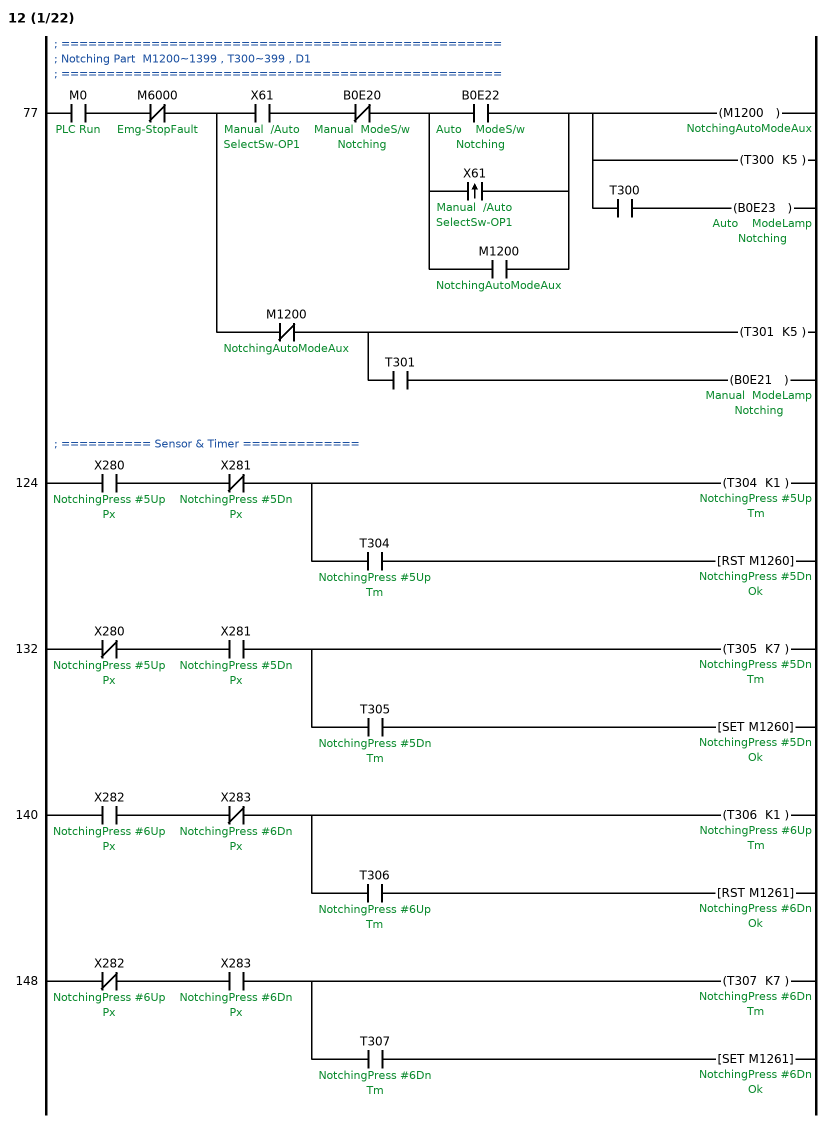
; =================================================
; Notching Part  M1200~1399 , T300~399 , D1
; =================================================
77    LD      M0  ; PLC Run
      ANI     M6000  ; Emg-StopFault
      MPS
      AND     X61  ; Manual  /Auto   SelectSw-OP1
      ANI     B0E20  ; Manual  ModeS/w Notching
      LD      B0E22  ; Auto    ModeS/w Notching
      ORP     X61  ; Manual  /Auto   SelectSw-OP1
      OR      M1200  ; NotchingAutoModeAux
      ANB
      OUT     M1200  ; NotchingAutoModeAux
      OUT     T300 K5
      AND     T300
      OUT     B0E23  ; Auto    ModeLampNotching
      MPP
      ANI     M1200  ; NotchingAutoModeAux
      OUT     T301 K5
      AND     T301
      OUT     B0E21  ; Manual  ModeLampNotching
; ========== Sensor & Timer =============
124   LD      X280  ; NotchingPress #5Up Px
      ANI     X281  ; NotchingPress #5Dn Px
      OUT     T304 K1  ; NotchingPress #5Up Tm
      AND     T304  ; NotchingPress #5Up Tm
      RST     M1260  ; NotchingPress #5Dn Ok
132   LDI     X280  ; NotchingPress #5Up Px
      AND     X281  ; NotchingPress #5Dn Px
      OUT     T305 K7  ; NotchingPress #5Dn Tm
      AND     T305  ; NotchingPress #5Dn Tm
      SET     M1260  ; NotchingPress #5Dn Ok
140   LD      X282  ; NotchingPress #6Up Px
      ANI     X283  ; NotchingPress #6Dn Px
      OUT     T306 K1  ; NotchingPress #6Up Tm
      AND     T306  ; NotchingPress #6Up Tm
      RST     M1261  ; NotchingPress #6Dn Ok
148   LDI     X282  ; NotchingPress #6Up Px
      AND     X283  ; NotchingPress #6Dn Px
      OUT     T307 K7  ; NotchingPress #6Dn Tm
      AND     T307  ; NotchingPress #6Dn Tm
      SET     M1261  ; NotchingPress #6Dn Ok
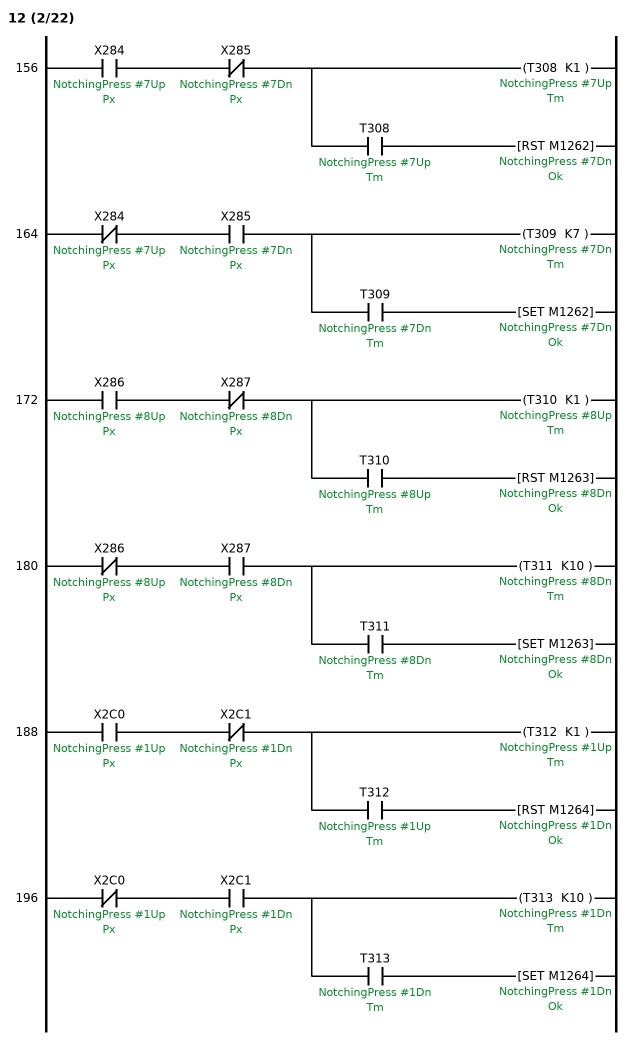
156   LD      X284  ; NotchingPress #7Up Px
      ANI     X285  ; NotchingPress #7Dn Px
      OUT     T308 K1  ; NotchingPress #7Up Tm
      AND     T308  ; NotchingPress #7Up Tm
      RST     M1262  ; NotchingPress #7Dn Ok
164   LDI     X284  ; NotchingPress #7Up Px
      AND     X285  ; NotchingPress #7Dn Px
      OUT     T309 K7  ; NotchingPress #7Dn Tm
      AND     T309  ; NotchingPress #7Dn Tm
      SET     M1262  ; NotchingPress #7Dn Ok
172   LD      X286  ; NotchingPress #8Up Px
      ANI     X287  ; NotchingPress #8Dn Px
      OUT     T310 K1  ; NotchingPress #8Up Tm
      AND     T310  ; NotchingPress #8Up Tm
      RST     M1263  ; NotchingPress #8Dn Ok
180   LDI     X286  ; NotchingPress #8Up Px
      AND     X287  ; NotchingPress #8Dn Px
      OUT     T311 K10  ; NotchingPress #8Dn Tm
      AND     T311  ; NotchingPress #8Dn Tm
      SET     M1263  ; NotchingPress #8Dn Ok
188   LD      X2C0  ; NotchingPress #1Up Px
      ANI     X2C1  ; NotchingPress #1Dn Px
      OUT     T312 K1  ; NotchingPress #1Up Tm
      AND     T312  ; NotchingPress #1Up Tm
      RST     M1264  ; NotchingPress #1Dn Ok
196   LDI     X2C0  ; NotchingPress #1Up Px
      AND     X2C1  ; NotchingPress #1Dn Px
      OUT     T313 K10  ; NotchingPress #1Dn Tm
      AND     T313  ; NotchingPress #1Dn Tm
      SET     M1264  ; NotchingPress #1Dn Ok
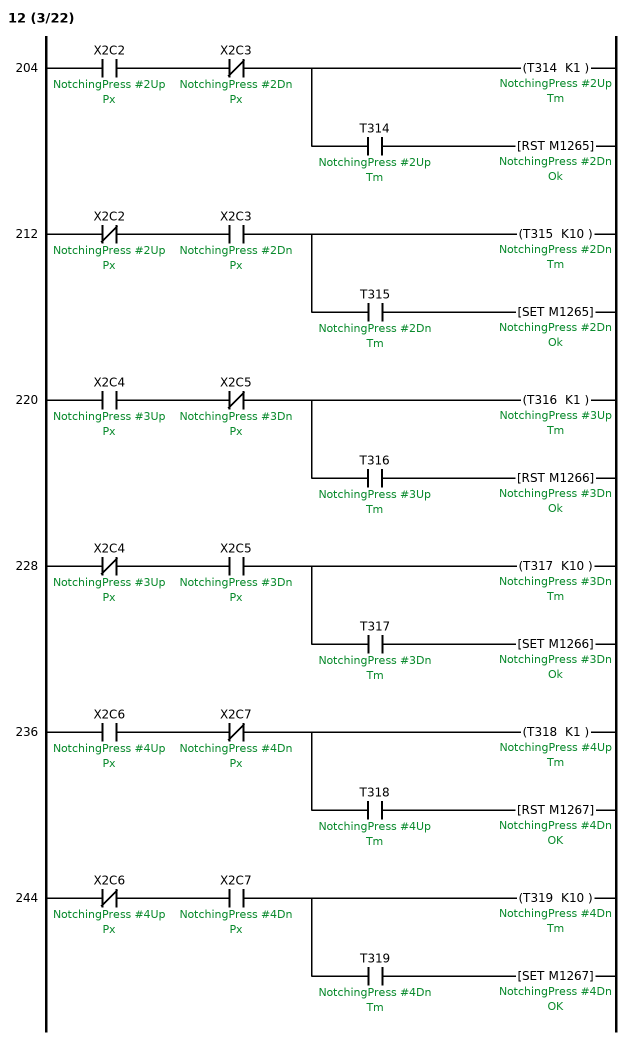
204   LD      X2C2  ; NotchingPress #2Up Px
      ANI     X2C3  ; NotchingPress #2Dn Px
      OUT     T314 K1  ; NotchingPress #2Up Tm
      AND     T314  ; NotchingPress #2Up Tm
      RST     M1265  ; NotchingPress #2Dn Ok
212   LDI     X2C2  ; NotchingPress #2Up Px
      AND     X2C3  ; NotchingPress #2Dn Px
      OUT     T315 K10  ; NotchingPress #2Dn Tm
      AND     T315  ; NotchingPress #2Dn Tm
      SET     M1265  ; NotchingPress #2Dn Ok
220   LD      X2C4  ; NotchingPress #3Up Px
      ANI     X2C5  ; NotchingPress #3Dn Px
      OUT     T316 K1  ; NotchingPress #3Up Tm
      AND     T316  ; NotchingPress #3Up Tm
      RST     M1266  ; NotchingPress #3Dn Ok
228   LDI     X2C4  ; NotchingPress #3Up Px
      AND     X2C5  ; NotchingPress #3Dn Px
      OUT     T317 K10  ; NotchingPress #3Dn Tm
      AND     T317  ; NotchingPress #3Dn Tm
      SET     M1266  ; NotchingPress #3Dn Ok
236   LD      X2C6  ; NotchingPress #4Up Px
      ANI     X2C7  ; NotchingPress #4Dn Px
      OUT     T318 K1  ; NotchingPress #4Up Tm
      AND     T318  ; NotchingPress #4Up Tm
      RST     M1267  ; NotchingPress #4Dn OK
244   LDI     X2C6  ; NotchingPress #4Up Px
      AND     X2C7  ; NotchingPress #4Dn Px
      OUT     T319 K10  ; NotchingPress #4Dn Tm
      AND     T319  ; NotchingPress #4Dn Tm
      SET     M1267  ; NotchingPress #4Dn OK
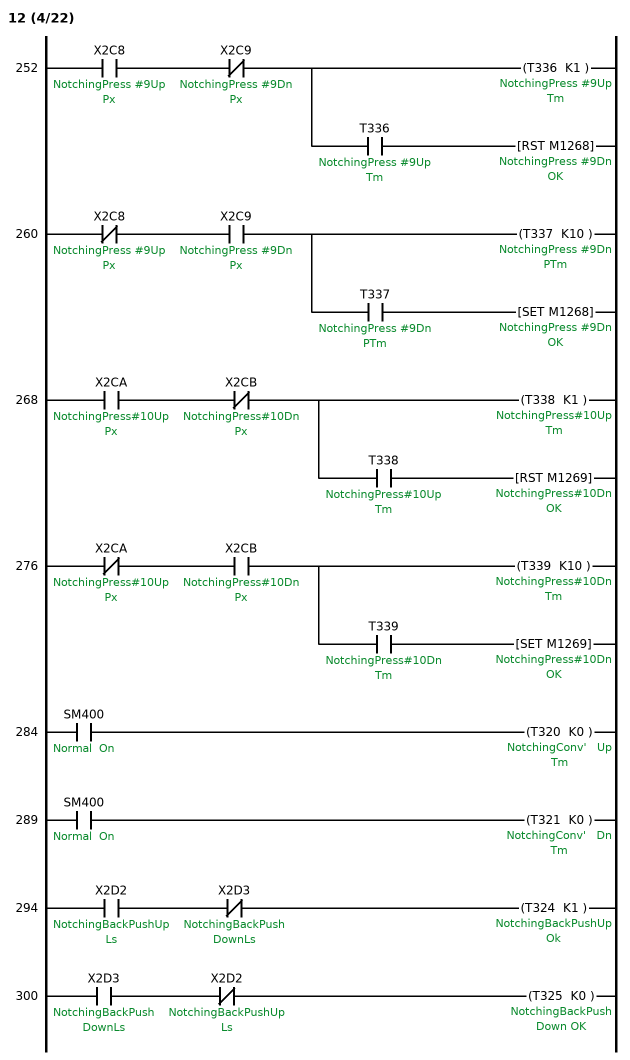
252   LD      X2C8  ; NotchingPress #9Up Px
      ANI     X2C9  ; NotchingPress #9Dn Px
      OUT     T336 K1  ; NotchingPress #9Up Tm
      AND     T336  ; NotchingPress #9Up Tm
      RST     M1268  ; NotchingPress #9Dn OK
260   LDI     X2C8  ; NotchingPress #9Up Px
      AND     X2C9  ; NotchingPress #9Dn Px
      OUT     T337 K10  ; NotchingPress #9Dn PTm
      AND     T337  ; NotchingPress #9Dn PTm
      SET     M1268  ; NotchingPress #9Dn OK
268   LD      X2CA  ; NotchingPress#10Up Px
      ANI     X2CB  ; NotchingPress#10Dn Px
      OUT     T338 K1  ; NotchingPress#10Up Tm
      AND     T338  ; NotchingPress#10Up Tm
      RST     M1269  ; NotchingPress#10Dn OK
276   LDI     X2CA  ; NotchingPress#10Up Px
      AND     X2CB  ; NotchingPress#10Dn Px
      OUT     T339 K10  ; NotchingPress#10Dn Tm
      AND     T339  ; NotchingPress#10Dn Tm
      SET     M1269  ; NotchingPress#10Dn OK
284   LD      SM400  ; Normal  On
      OUT     T320 K0  ; NotchingConv'   Up Tm
289   LD      SM400  ; Normal  On
      OUT     T321 K0  ; NotchingConv'   Dn Tm
294   LD      X2D2  ; NotchingBackPushUpLs
      ANI     X2D3  ; NotchingBackPushDownLs
      OUT     T324 K1  ; NotchingBackPushUp Ok
300   LD      X2D3  ; NotchingBackPushDownLs
      ANI     X2D2  ; NotchingBackPushUpLs
      OUT     T325 K0  ; NotchingBackPushDown OK
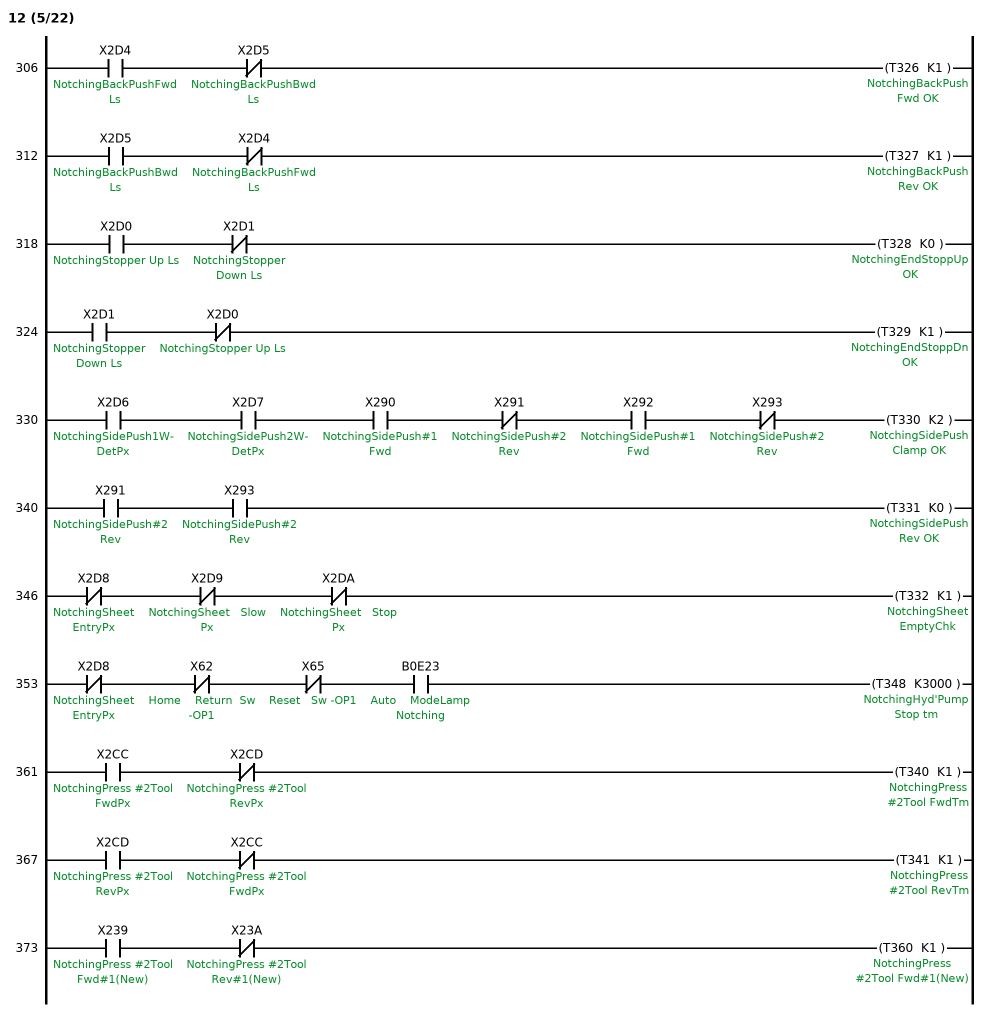
306   LD      X2D4  ; NotchingBackPushFwdLs
      ANI     X2D5  ; NotchingBackPushBwdLs
      OUT     T326 K1  ; NotchingBackPushFwd OK
312   LD      X2D5  ; NotchingBackPushBwdLs
      ANI     X2D4  ; NotchingBackPushFwdLs
      OUT     T327 K1  ; NotchingBackPushRev OK
318   LD      X2D0  ; NotchingStopper Up Ls
      ANI     X2D1  ; NotchingStopper Down Ls
      OUT     T328 K0  ; NotchingEndStoppUp OK
324   LD      X2D1  ; NotchingStopper Down Ls
      ANI     X2D0  ; NotchingStopper Up Ls
      OUT     T329 K1  ; NotchingEndStoppDn OK
330   LD      X2D6  ; NotchingSidePush1W-DetPx
      AND     X2D7  ; NotchingSidePush2W-DetPx
      AND     X290  ; NotchingSidePush#1 Fwd
      ANI     X291  ; NotchingSidePush#2 Rev
      AND     X292  ; NotchingSidePush#1 Fwd
      ANI     X293  ; NotchingSidePush#2 Rev
      OUT     T330 K2  ; NotchingSidePushClamp OK
340   LD      X291  ; NotchingSidePush#2 Rev
      AND     X293  ; NotchingSidePush#2 Rev
      OUT     T331 K0  ; NotchingSidePushRev OK
346   LDI     X2D8  ; NotchingSheet   EntryPx
      ANI     X2D9  ; NotchingSheet   Slow Px
      ANI     X2DA  ; NotchingSheet   Stop Px
      OUT     T332 K1  ; NotchingSheet   EmptyChk
353   LDI     X2D8  ; NotchingSheet   EntryPx
      ANI     X62  ; Home    Return  Sw -OP1
      ANI     X65  ; Reset   Sw -OP1
      AND     B0E23  ; Auto    ModeLampNotching
      OUT     T348 K3000  ; NotchingHyd'PumpStop tm
361   LD      X2CC  ; NotchingPress #2Tool FwdPx
      ANI     X2CD  ; NotchingPress #2Tool RevPx
      OUT     T340 K1  ; NotchingPress #2Tool FwdTm
367   LD      X2CD  ; NotchingPress #2Tool RevPx
      ANI     X2CC  ; NotchingPress #2Tool FwdPx
      OUT     T341 K1  ; NotchingPress #2Tool RevTm
373   LD      X239  ; NotchingPress #2Tool Fwd#1(New)
      ANI     X23A  ; NotchingPress #2Tool Rev#1(New)
      OUT     T360 K1  ; NotchingPress #2Tool Fwd#1(New)
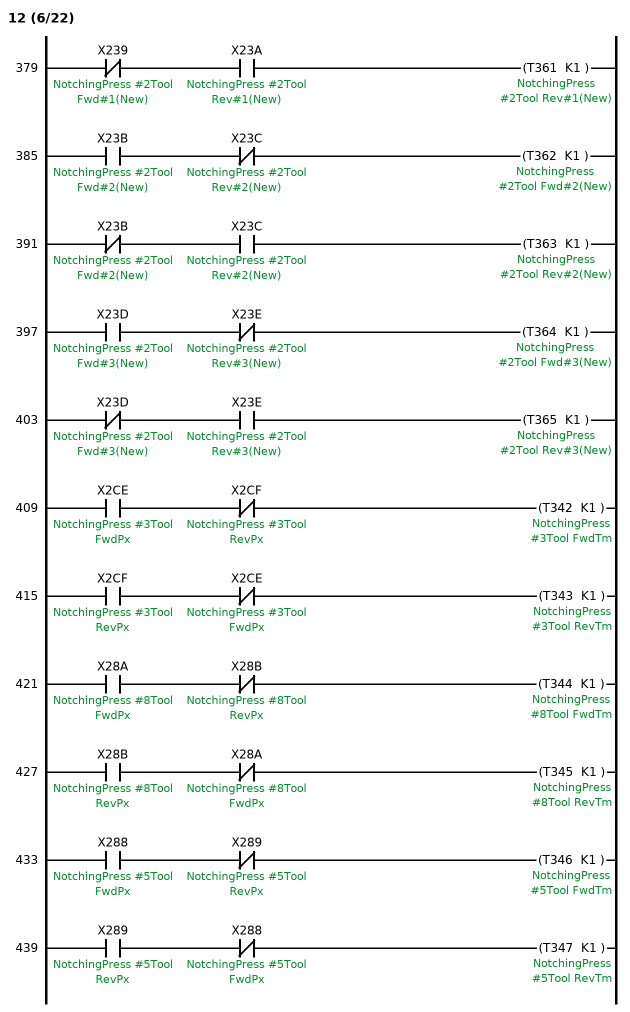
379   LDI     X239  ; NotchingPress #2Tool Fwd#1(New)
      AND     X23A  ; NotchingPress #2Tool Rev#1(New)
      OUT     T361 K1  ; NotchingPress #2Tool Rev#1(New)
385   LD      X23B  ; NotchingPress #2Tool Fwd#2(New)
      ANI     X23C  ; NotchingPress #2Tool Rev#2(New)
      OUT     T362 K1  ; NotchingPress #2Tool Fwd#2(New)
391   LDI     X23B  ; NotchingPress #2Tool Fwd#2(New)
      AND     X23C  ; NotchingPress #2Tool Rev#2(New)
      OUT     T363 K1  ; NotchingPress #2Tool Rev#2(New)
397   LD      X23D  ; NotchingPress #2Tool Fwd#3(New)
      ANI     X23E  ; NotchingPress #2Tool Rev#3(New)
      OUT     T364 K1  ; NotchingPress #2Tool Fwd#3(New)
403   LDI     X23D  ; NotchingPress #2Tool Fwd#3(New)
      AND     X23E  ; NotchingPress #2Tool Rev#3(New)
      OUT     T365 K1  ; NotchingPress #2Tool Rev#3(New)
409   LD      X2CE  ; NotchingPress #3Tool FwdPx
      ANI     X2CF  ; NotchingPress #3Tool RevPx
      OUT     T342 K1  ; NotchingPress #3Tool FwdTm
415   LD      X2CF  ; NotchingPress #3Tool RevPx
      ANI     X2CE  ; NotchingPress #3Tool FwdPx
      OUT     T343 K1  ; NotchingPress #3Tool RevTm
421   LD      X28A  ; NotchingPress #8Tool FwdPx
      ANI     X28B  ; NotchingPress #8Tool RevPx
      OUT     T344 K1  ; NotchingPress #8Tool FwdTm
427   LD      X28B  ; NotchingPress #8Tool RevPx
      ANI     X28A  ; NotchingPress #8Tool FwdPx
      OUT     T345 K1  ; NotchingPress #8Tool RevTm
433   LD      X288  ; NotchingPress #5Tool FwdPx
      ANI     X289  ; NotchingPress #5Tool RevPx
      OUT     T346 K1  ; NotchingPress #5Tool FwdTm
439   LD      X289  ; NotchingPress #5Tool RevPx
      ANI     X288  ; NotchingPress #5Tool FwdPx
      OUT     T347 K1  ; NotchingPress #5Tool RevTm
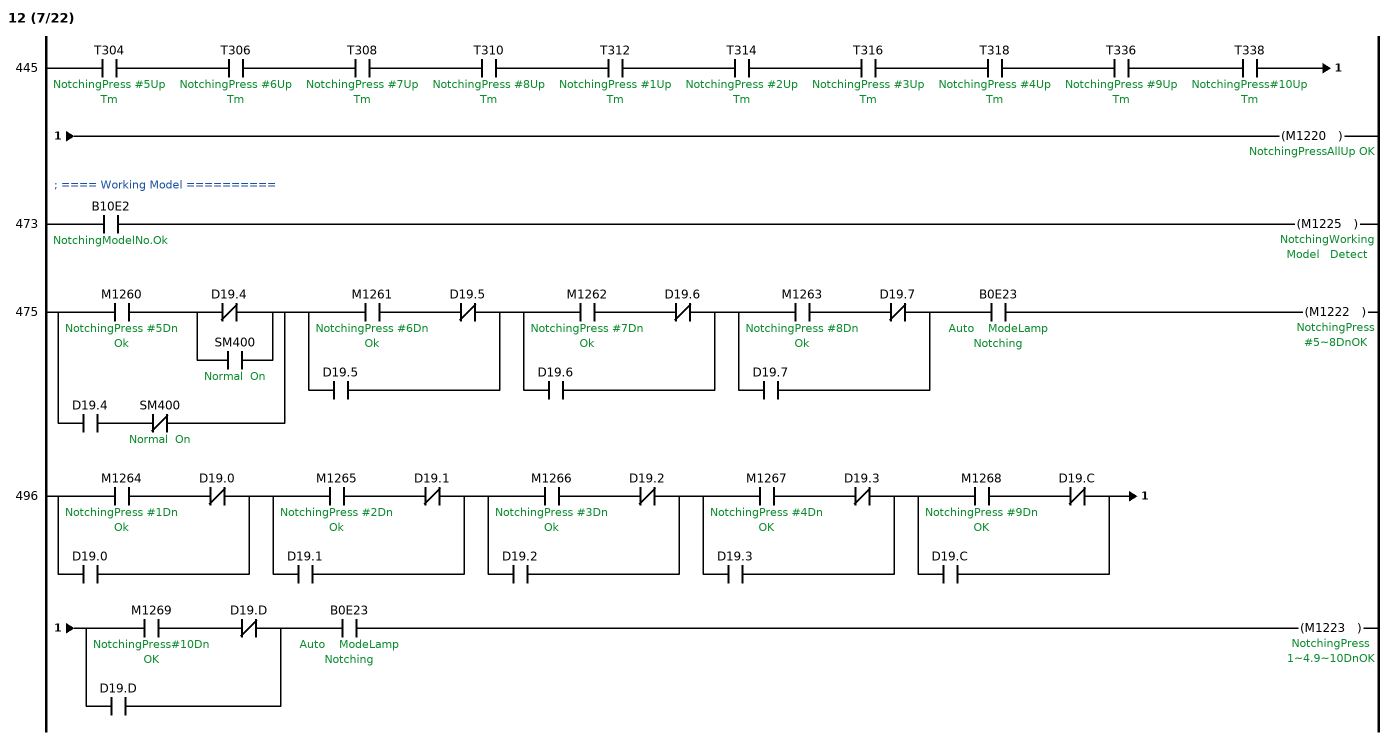
445   LD      T304  ; NotchingPress #5Up Tm
      AND     T306  ; NotchingPress #6Up Tm
      AND     T308  ; NotchingPress #7Up Tm
      AND     T310  ; NotchingPress #8Up Tm
      AND     T312  ; NotchingPress #1Up Tm
      AND     T314  ; NotchingPress #2Up Tm
      AND     T316  ; NotchingPress #3Up Tm
      AND     T318  ; NotchingPress #4Up Tm
      AND     T336  ; NotchingPress #9Up Tm
      AND     T338  ; NotchingPress#10Up Tm
      OUT     M1220  ; NotchingPressAllUp OK
; ==== Working Model ==========
473   LD      B10E2  ; NotchingModelNo.Ok
      OUT     M1225  ; NotchingWorking Model   Detect
475   LD      M1260  ; NotchingPress #5Dn Ok
      LDI     D19.4
      OR      SM400  ; Normal  On
      ANB
      LD      D19.4
      ANI     SM400  ; Normal  On
      ORB
      LD      M1261  ; NotchingPress #6Dn Ok
      ANI     D19.5
      OR      D19.5
      ANB
      LD      M1262  ; NotchingPress #7Dn Ok
      ANI     D19.6
      OR      D19.6
      ANB
      LD      M1263  ; NotchingPress #8Dn Ok
      ANI     D19.7
      OR      D19.7
      ANB
      AND     B0E23  ; Auto    ModeLampNotching
      OUT     M1222  ; NotchingPress   #5~8DnOK
496   LD      M1264  ; NotchingPress #1Dn Ok
      ANI     D19.0
      OR      D19.0
      LD      M1265  ; NotchingPress #2Dn Ok
      ANI     D19.1
      OR      D19.1
      ANB
      LD      M1266  ; NotchingPress #3Dn Ok
      ANI     D19.2
      OR      D19.2
      ANB
      LD      M1267  ; NotchingPress #4Dn OK
      ANI     D19.3
      OR      D19.3
      ANB
      LD      M1268  ; NotchingPress #9Dn OK
      ANI     D19.C
      OR      D19.C
      ANB
      LD      M1269  ; NotchingPress#10Dn OK
      ANI     D19.D
      OR      D19.D
      ANB
      AND     B0E23  ; Auto    ModeLampNotching
      OUT     M1223  ; NotchingPress   1~4.9~10DnOK
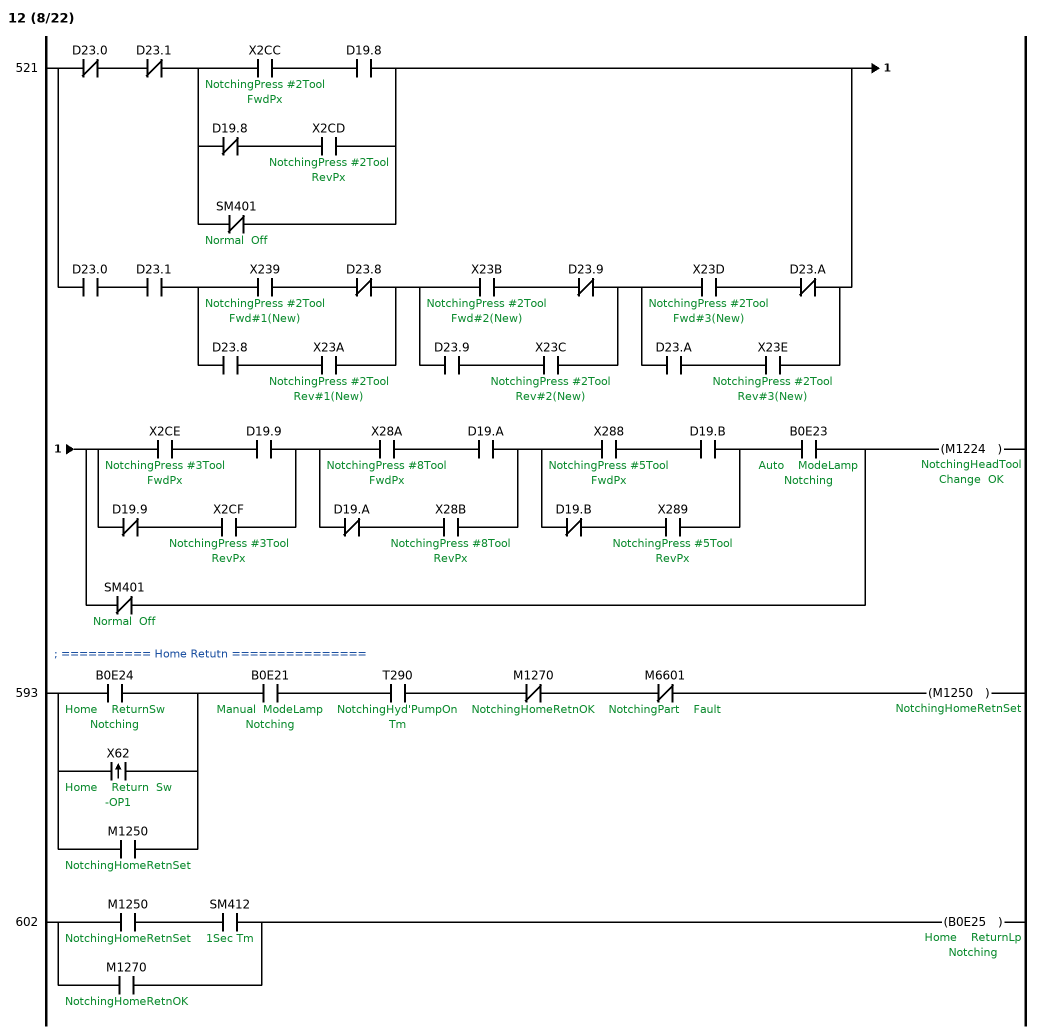
521   LDI     D23.0
      ANI     D23.1
      LD      X2CC  ; NotchingPress #2Tool FwdPx
      AND     D19.8
      LDI     D19.8
      AND     X2CD  ; NotchingPress #2Tool RevPx
      ORB
      ORI     SM401  ; Normal  Off
      ANB
      LD      D23.0
      AND     D23.1
      LD      X239  ; NotchingPress #2Tool Fwd#1(New)
      ANI     D23.8
      LD      D23.8
      AND     X23A  ; NotchingPress #2Tool Rev#1(New)
      ORB
      ANB
      LD      X23B  ; NotchingPress #2Tool Fwd#2(New)
      ANI     D23.9
      LD      D23.9
      AND     X23C  ; NotchingPress #2Tool Rev#2(New)
      ORB
      ANB
      LD      X23D  ; NotchingPress #2Tool Fwd#3(New)
      ANI     D23.A
      LD      D23.A
      AND     X23E  ; NotchingPress #2Tool Rev#3(New)
      ORB
      ANB
      ORB
      LD      X2CE  ; NotchingPress #3Tool FwdPx
      AND     D19.9
      LDI     D19.9
      AND     X2CF  ; NotchingPress #3Tool RevPx
      ORB
      LD      X28A  ; NotchingPress #8Tool FwdPx
      AND     D19.A
      LDI     D19.A
      AND     X28B  ; NotchingPress #8Tool RevPx
      ORB
      ANB
      LD      X288  ; NotchingPress #5Tool FwdPx
      AND     D19.B
      LDI     D19.B
      AND     X289  ; NotchingPress #5Tool RevPx
      ORB
      ANB
      AND     B0E23  ; Auto    ModeLampNotching
      ORI     SM401  ; Normal  Off
      ANB
      OUT     M1224  ; NotchingHeadToolChange  OK
; ========== Home Retutn ===============
593   LD      B0E24  ; Home    ReturnSwNotching
      ORP     X62  ; Home    Return  Sw -OP1
      OR      M1250  ; NotchingHomeRetnSet
      AND     B0E21  ; Manual  ModeLampNotching
      AND     T290  ; NotchingHyd'PumpOn Tm
      ANI     M1270  ; NotchingHomeRetnOK
      ANI     M6601  ; NotchingPart    Fault
      OUT     M1250  ; NotchingHomeRetnSet
602   LD      M1250  ; NotchingHomeRetnSet
      AND     SM412  ; 1Sec Tm
      OR      M1270  ; NotchingHomeRetnOK
      OUT     B0E25  ; Home    ReturnLpNotching
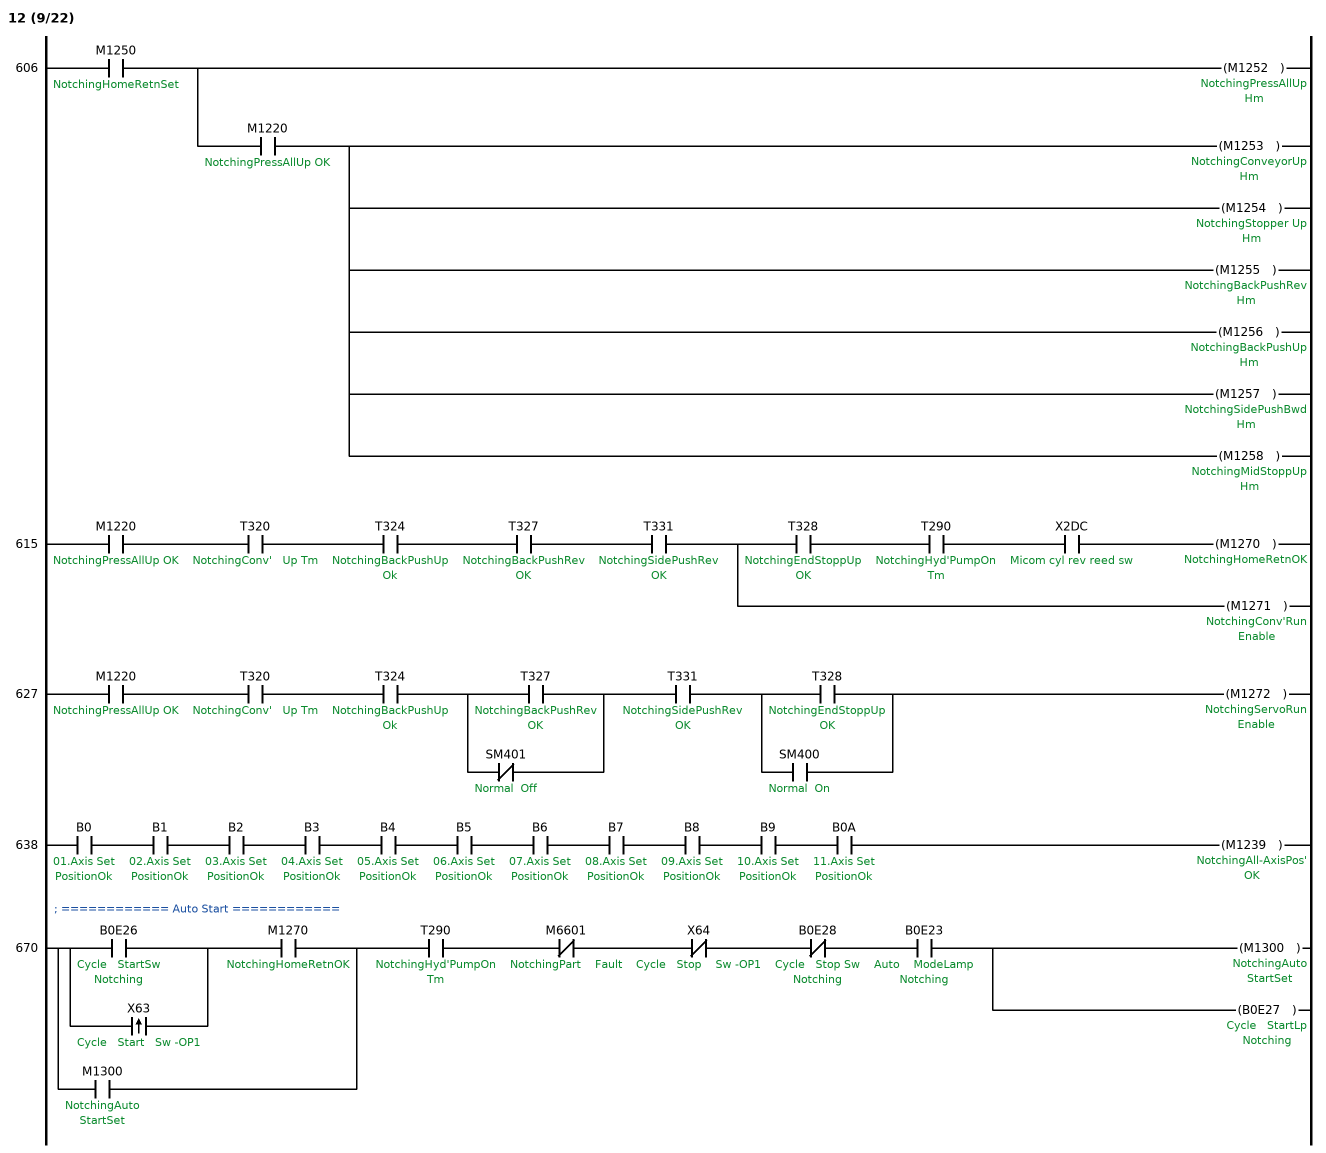
606   LD      M1250  ; NotchingHomeRetnSet
      OUT     M1252  ; NotchingPressAllUp Hm
      AND     M1220  ; NotchingPressAllUp OK
      OUT     M1253  ; NotchingConveyorUp Hm
      OUT     M1254  ; NotchingStopper Up Hm
      OUT     M1255  ; NotchingBackPushRev Hm
      OUT     M1256  ; NotchingBackPushUp Hm
      OUT     M1257  ; NotchingSidePushBwd Hm
      OUT     M1258  ; NotchingMidStoppUp Hm
615   LD      M1220  ; NotchingPressAllUp OK
      AND     T320  ; NotchingConv'   Up Tm
      AND     T324  ; NotchingBackPushUp Ok
      AND     T327  ; NotchingBackPushRev OK
      AND     T331  ; NotchingSidePushRev OK
      MPS
      AND     T328  ; NotchingEndStoppUp OK
      AND     T290  ; NotchingHyd'PumpOn Tm
      AND     X2DC  ; Micom cyl rev reed sw
      OUT     M1270  ; NotchingHomeRetnOK
      MPP
      OUT     M1271  ; NotchingConv'RunEnable
627   LD      M1220  ; NotchingPressAllUp OK
      AND     T320  ; NotchingConv'   Up Tm
      AND     T324  ; NotchingBackPushUp Ok
      LD      T327  ; NotchingBackPushRev OK
      ORI     SM401  ; Normal  Off
      ANB
      AND     T331  ; NotchingSidePushRev OK
      LD      T328  ; NotchingEndStoppUp OK
      OR      SM400  ; Normal  On
      ANB
      OUT     M1272  ; NotchingServoRunEnable
638   LD      B0  ; 01.Axis Set     PositionOk
      AND     B1  ; 02.Axis Set     PositionOk
      AND     B2  ; 03.Axis Set     PositionOk
      AND     B3  ; 04.Axis Set     PositionOk
      AND     B4  ; 05.Axis Set     PositionOk
      AND     B5  ; 06.Axis Set     PositionOk
      AND     B6  ; 07.Axis Set     PositionOk
      AND     B7  ; 08.Axis Set     PositionOk
      AND     B8  ; 09.Axis Set     PositionOk
      AND     B9  ; 10.Axis Set     PositionOk
      AND     B0A  ; 11.Axis Set     PositionOk
      OUT     M1239  ; NotchingAll-AxisPos' OK
; ============ Auto Start ============
670   LD      B0E26  ; Cycle   StartSw Notching
      ORP     X63  ; Cycle   Start   Sw -OP1
      AND     M1270  ; NotchingHomeRetnOK
      OR      M1300  ; NotchingAuto    StartSet
      AND     T290  ; NotchingHyd'PumpOn Tm
      ANI     M6601  ; NotchingPart    Fault
      ANI     X64  ; Cycle   Stop    Sw -OP1
      ANI     B0E28  ; Cycle   Stop Sw Notching
      AND     B0E23  ; Auto    ModeLampNotching
      OUT     M1300  ; NotchingAuto    StartSet
      OUT     B0E27  ; Cycle   StartLp Notching
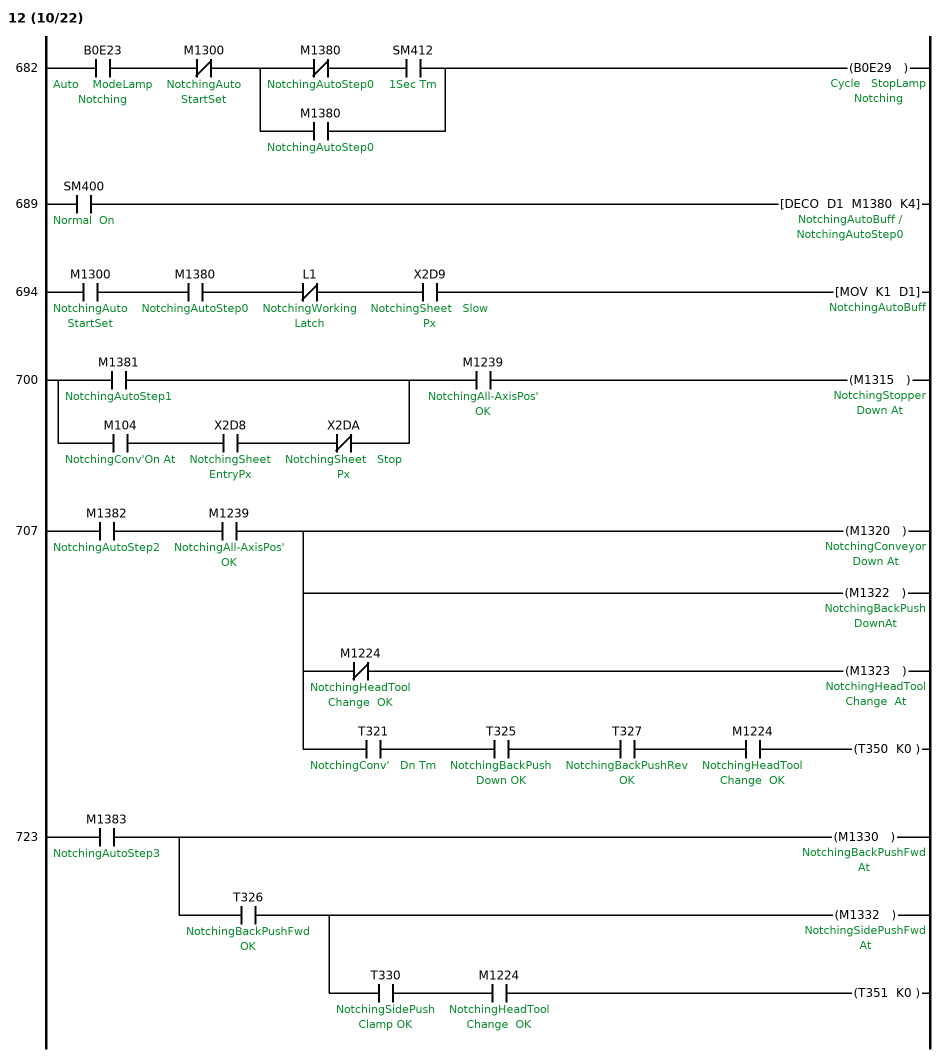
682   LD      B0E23  ; Auto    ModeLampNotching
      ANI     M1300  ; NotchingAuto    StartSet
      LDI     M1380  ; NotchingAutoStep0
      AND     SM412  ; 1Sec Tm
      OR      M1380  ; NotchingAutoStep0
      ANB
      OUT     B0E29  ; Cycle   StopLampNotching
689   LD      SM400  ; Normal  On
      DECO    D1 M1380 K4  ; NotchingAutoBuff
694   LD      M1300  ; NotchingAuto    StartSet
      AND     M1380  ; NotchingAutoStep0
      ANI     L1  ; NotchingWorking Latch
      AND     X2D9  ; NotchingSheet   Slow Px
      MOV     K1 D1
700   LD      M1381  ; NotchingAutoStep1
      LD      M104  ; NotchingConv'On At
      AND     X2D8  ; NotchingSheet   EntryPx
      ANI     X2DA  ; NotchingSheet   Stop Px
      ORB
      AND     M1239  ; NotchingAll-AxisPos' OK
      OUT     M1315  ; NotchingStopper Down At
707   LD      M1382  ; NotchingAutoStep2
      AND     M1239  ; NotchingAll-AxisPos' OK
      OUT     M1320  ; NotchingConveyorDown At
      OUT     M1322  ; NotchingBackPushDownAt
      MPS
      ANI     M1224  ; NotchingHeadToolChange  OK
      OUT     M1323  ; NotchingHeadToolChange  At
      MPP
      AND     T321  ; NotchingConv'   Dn Tm
      AND     T325  ; NotchingBackPushDown OK
      AND     T327  ; NotchingBackPushRev OK
      AND     M1224  ; NotchingHeadToolChange  OK
      OUT     T350 K0
723   LD      M1383  ; NotchingAutoStep3
      OUT     M1330  ; NotchingBackPushFwdAt
      AND     T326  ; NotchingBackPushFwd OK
      OUT     M1332  ; NotchingSidePushFwdAt
      AND     T330  ; NotchingSidePushClamp OK
      AND     M1224  ; NotchingHeadToolChange  OK
      OUT     T351 K0
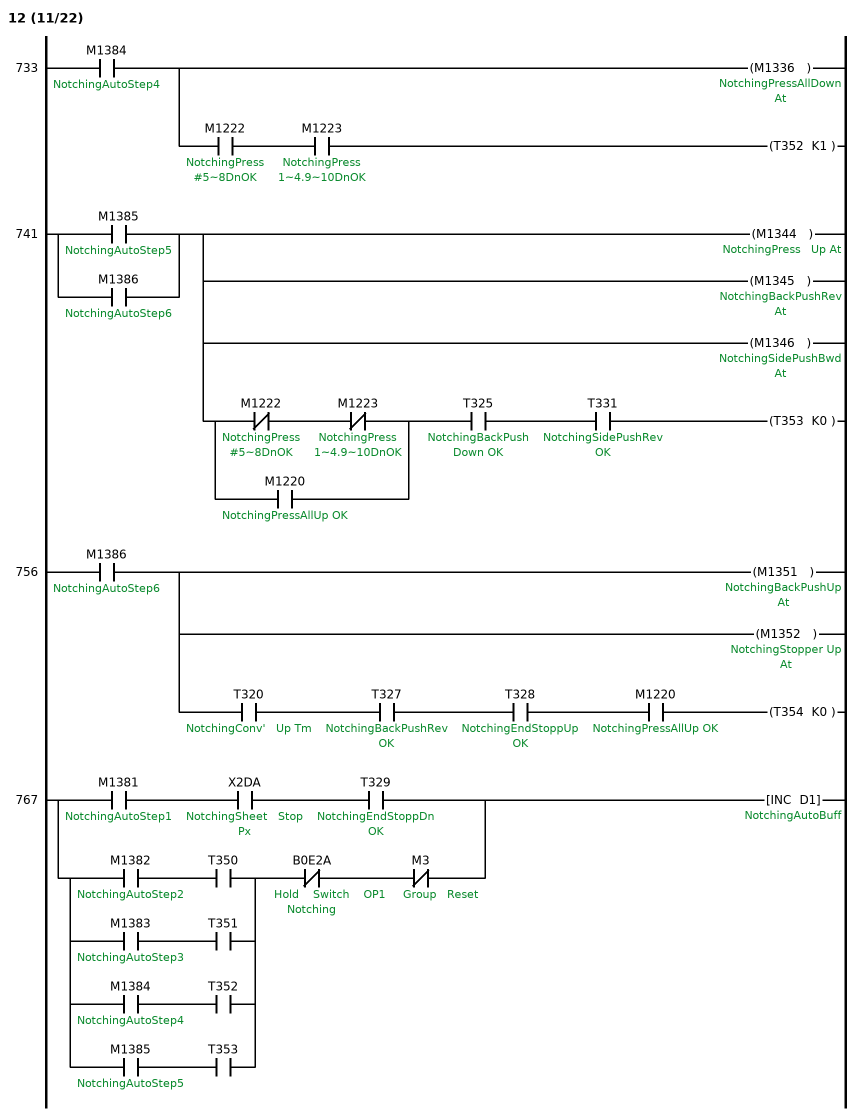
733   LD      M1384  ; NotchingAutoStep4
      OUT     M1336  ; NotchingPressAllDown At
      AND     M1222  ; NotchingPress   #5~8DnOK
      AND     M1223  ; NotchingPress   1~4.9~10DnOK
      OUT     T352 K1
741   LD      M1385  ; NotchingAutoStep5
      OR      M1386  ; NotchingAutoStep6
      OUT     M1344  ; NotchingPress   Up At
      OUT     M1345  ; NotchingBackPushRev At
      OUT     M1346  ; NotchingSidePushBwd At
      LDI     M1222  ; NotchingPress   #5~8DnOK
      ANI     M1223  ; NotchingPress   1~4.9~10DnOK
      OR      M1220  ; NotchingPressAllUp OK
      ANB
      AND     T325  ; NotchingBackPushDown OK
      AND     T331  ; NotchingSidePushRev OK
      OUT     T353 K0
756   LD      M1386  ; NotchingAutoStep6
      OUT     M1351  ; NotchingBackPushUp At
      OUT     M1352  ; NotchingStopper Up At
      AND     T320  ; NotchingConv'   Up Tm
      AND     T327  ; NotchingBackPushRev OK
      AND     T328  ; NotchingEndStoppUp OK
      AND     M1220  ; NotchingPressAllUp OK
      OUT     T354 K0
767   LD      M1381  ; NotchingAutoStep1
      AND     X2DA  ; NotchingSheet   Stop Px
      AND     T329  ; NotchingEndStoppDn OK
      LD      M1382  ; NotchingAutoStep2
      AND     T350
      LD      M1383  ; NotchingAutoStep3
      AND     T351
      ORB
      LD      M1384  ; NotchingAutoStep4
      AND     T352
      ORB
      LD      M1385  ; NotchingAutoStep5
      AND     T353
      ORB
      ANI     B0E2A  ; Hold    Switch  Notching
      ANI     M3  ; OP1     Group   Reset
      ORB
      INC     D1
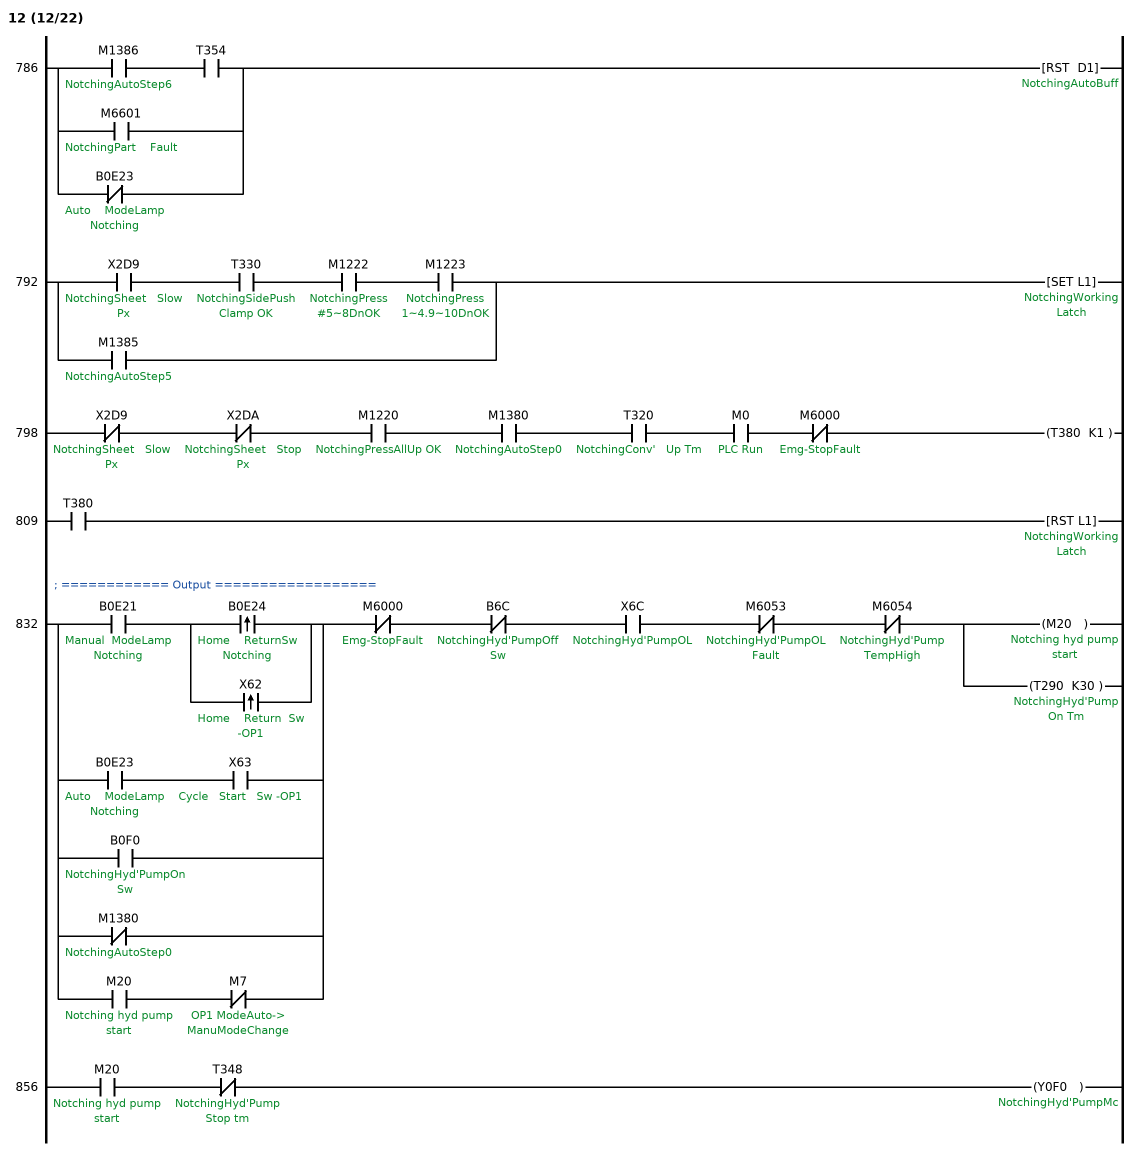
786   LD      M1386  ; NotchingAutoStep6
      AND     T354
      OR      M6601  ; NotchingPart    Fault
      ORI     B0E23  ; Auto    ModeLampNotching
      RST     D1  ; NotchingAutoBuff
792   LD      X2D9  ; NotchingSheet   Slow Px
      AND     T330  ; NotchingSidePushClamp OK
      AND     M1222  ; NotchingPress   #5~8DnOK
      AND     M1223  ; NotchingPress   1~4.9~10DnOK
      OR      M1385  ; NotchingAutoStep5
      SET     L1  ; NotchingWorking Latch
798   LDI     X2D9  ; NotchingSheet   Slow Px
      ANI     X2DA  ; NotchingSheet   Stop Px
      AND     M1220  ; NotchingPressAllUp OK
      AND     M1380  ; NotchingAutoStep0
      AND     T320  ; NotchingConv'   Up Tm
      AND     M0  ; PLC Run
      ANI     M6000  ; Emg-StopFault
      OUT     T380 K1
809   LD      T380
      RST     L1  ; NotchingWorking Latch
; ============ Output ==================
832   LD      B0E21  ; Manual  ModeLampNotching
      LDP     B0E24  ; Home    ReturnSwNotching
      ORP     X62  ; Home    Return  Sw -OP1
      ANB
      LD      B0E23  ; Auto    ModeLampNotching
      AND     X63  ; Cycle   Start   Sw -OP1
      ORB
      OR      B0F0  ; NotchingHyd'PumpOnSw
      ORI     M1380  ; NotchingAutoStep0
      LD      M20  ; Notching hyd pump start
      ANI     M7  ; OP1 ModeAuto->  ManuModeChange
      ORB
      ANI     M6000  ; Emg-StopFault
      ANI     B6C  ; NotchingHyd'PumpOffSw
      AND     X6C  ; NotchingHyd'PumpOL
      ANI     M6053  ; NotchingHyd'PumpOL Fault
      ANI     M6054  ; NotchingHyd'PumpTempHigh
      OUT     M20  ; Notching hyd pump start
      OUT     T290 K30  ; NotchingHyd'PumpOn Tm
856   LD      M20  ; Notching hyd pump start
      ANI     T348  ; NotchingHyd'PumpStop tm
      OUT     Y0F0  ; NotchingHyd'PumpMc
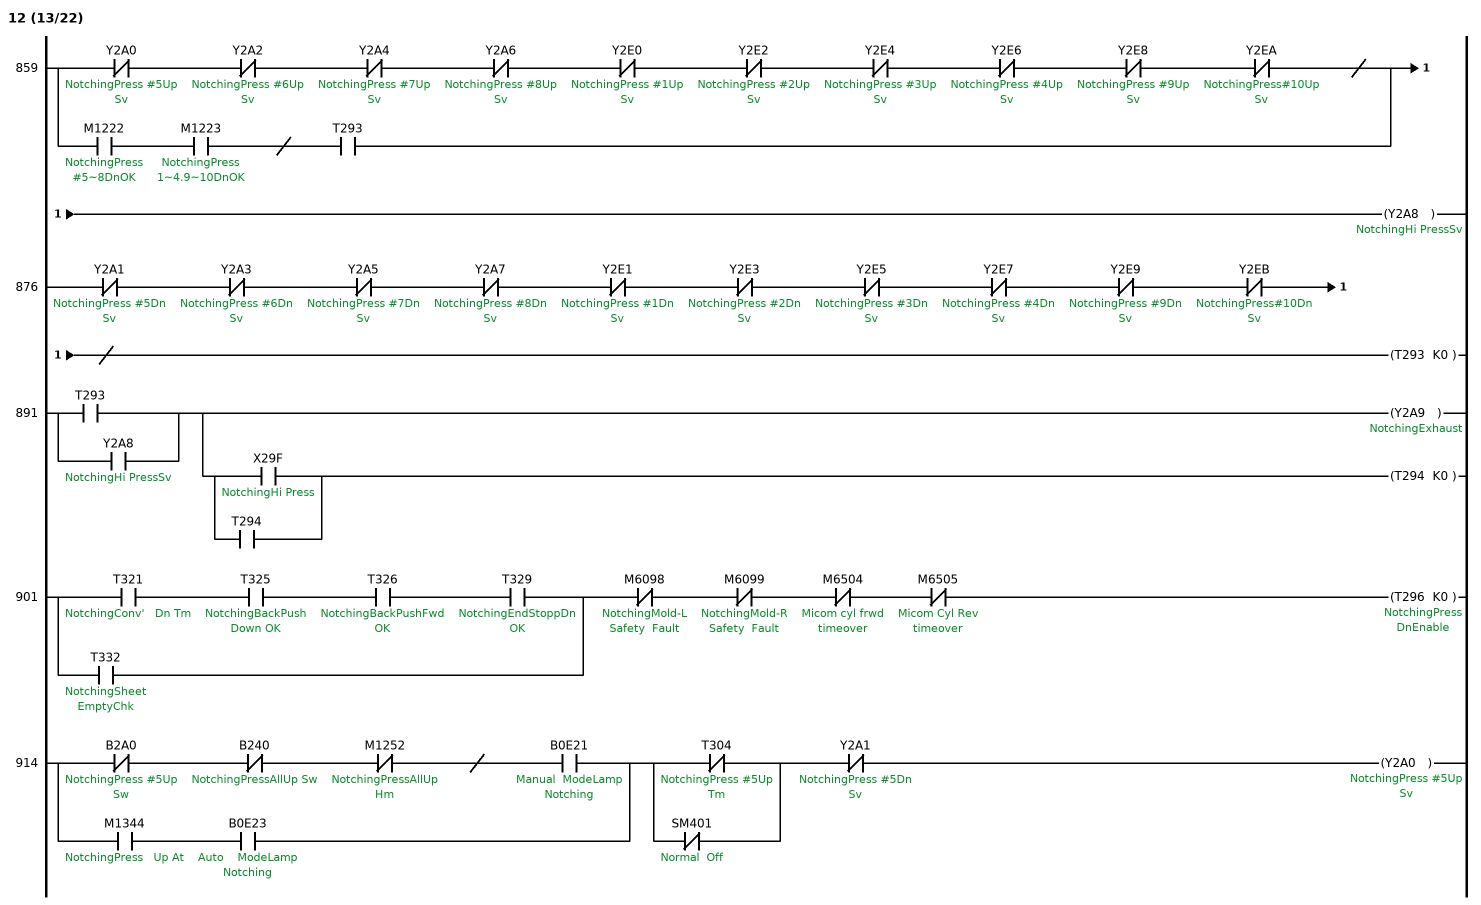
859   LDI     Y2A0  ; NotchingPress #5Up Sv
      ANI     Y2A2  ; NotchingPress #6Up Sv
      ANI     Y2A4  ; NotchingPress #7Up Sv
      ANI     Y2A6  ; NotchingPress #8Up Sv
      ANI     Y2E0  ; NotchingPress #1Up Sv
      ANI     Y2E2  ; NotchingPress #2Up Sv
      ANI     Y2E4  ; NotchingPress #3Up Sv
      ANI     Y2E6  ; NotchingPress #4Up Sv
      ANI     Y2E8  ; NotchingPress #9Up Sv
      ANI     Y2EA  ; NotchingPress#10Up Sv
      INV
      LD      M1222  ; NotchingPress   #5~8DnOK
      AND     M1223  ; NotchingPress   1~4.9~10DnOK
      INV
      AND     T293
      ORB
      OUT     Y2A8  ; NotchingHi PressSv
876   LDI     Y2A1  ; NotchingPress #5Dn Sv
      ANI     Y2A3  ; NotchingPress #6Dn Sv
      ANI     Y2A5  ; NotchingPress #7Dn Sv
      ANI     Y2A7  ; NotchingPress #8Dn Sv
      ANI     Y2E1  ; NotchingPress #1Dn Sv
      ANI     Y2E3  ; NotchingPress #2Dn Sv
      ANI     Y2E5  ; NotchingPress #3Dn Sv
      ANI     Y2E7  ; NotchingPress #4Dn Sv
      ANI     Y2E9  ; NotchingPress #9Dn Sv
      ANI     Y2EB  ; NotchingPress#10Dn Sv
      INV
      OUT     T293 K0
891   LD      T293
      OR      Y2A8  ; NotchingHi PressSv
      OUT     Y2A9  ; NotchingExhaust
      LD      X29F  ; NotchingHi Press
      OR      T294
      ANB
      OUT     T294 K0
901   LD      T321  ; NotchingConv'   Dn Tm
      AND     T325  ; NotchingBackPushDown OK
      AND     T326  ; NotchingBackPushFwd OK
      AND     T329  ; NotchingEndStoppDn OK
      OR      T332  ; NotchingSheet   EmptyChk
      ANI     M6098  ; NotchingMold-L  Safety  Fault
      ANI     M6099  ; NotchingMold-R  Safety  Fault
      ANI     M6504  ; Micom cyl frwd timeover
      ANI     M6505  ; Micom Cyl Rev timeover
      OUT     T296 K0  ; NotchingPress DnEnable
914   LDI     B2A0  ; NotchingPress #5Up Sw
      ANI     B240  ; NotchingPressAllUp Sw
      ANI     M1252  ; NotchingPressAllUp Hm
      INV
      AND     B0E21  ; Manual  ModeLampNotching
      LD      M1344  ; NotchingPress   Up At
      AND     B0E23  ; Auto    ModeLampNotching
      ORB
      LDI     T304  ; NotchingPress #5Up Tm
      ORI     SM401  ; Normal  Off
      ANB
      ANI     Y2A1  ; NotchingPress #5Dn Sv
      OUT     Y2A0  ; NotchingPress #5Up Sv
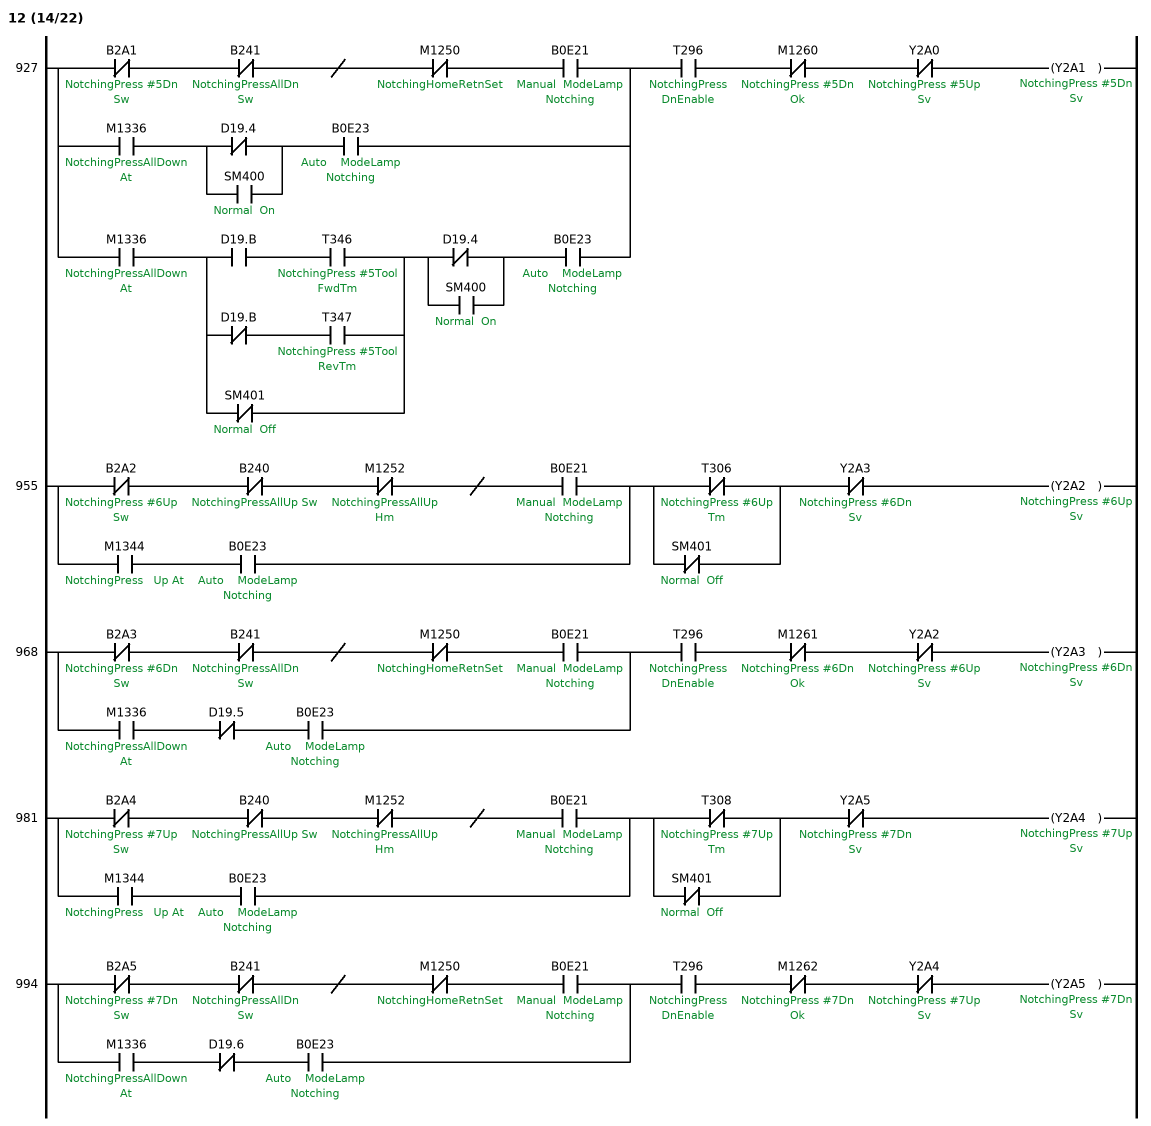
927   LDI     B2A1  ; NotchingPress #5Dn Sw
      ANI     B241  ; NotchingPressAllDn Sw
      INV
      ANI     M1250  ; NotchingHomeRetnSet
      AND     B0E21  ; Manual  ModeLampNotching
      LD      M1336  ; NotchingPressAllDown At
      LDI     D19.4
      OR      SM400  ; Normal  On
      ANB
      AND     B0E23  ; Auto    ModeLampNotching
      ORB
      LD      M1336  ; NotchingPressAllDown At
      LD      D19.B
      AND     T346  ; NotchingPress #5Tool FwdTm
      LDI     D19.B
      AND     T347  ; NotchingPress #5Tool RevTm
      ORB
      ORI     SM401  ; Normal  Off
      ANB
      LDI     D19.4
      OR      SM400  ; Normal  On
      ANB
      AND     B0E23  ; Auto    ModeLampNotching
      ORB
      AND     T296  ; NotchingPress DnEnable
      ANI     M1260  ; NotchingPress #5Dn Ok
      ANI     Y2A0  ; NotchingPress #5Up Sv
      OUT     Y2A1  ; NotchingPress #5Dn Sv
955   LDI     B2A2  ; NotchingPress #6Up Sw
      ANI     B240  ; NotchingPressAllUp Sw
      ANI     M1252  ; NotchingPressAllUp Hm
      INV
      AND     B0E21  ; Manual  ModeLampNotching
      LD      M1344  ; NotchingPress   Up At
      AND     B0E23  ; Auto    ModeLampNotching
      ORB
      LDI     T306  ; NotchingPress #6Up Tm
      ORI     SM401  ; Normal  Off
      ANB
      ANI     Y2A3  ; NotchingPress #6Dn Sv
      OUT     Y2A2  ; NotchingPress #6Up Sv
968   LDI     B2A3  ; NotchingPress #6Dn Sw
      ANI     B241  ; NotchingPressAllDn Sw
      INV
      ANI     M1250  ; NotchingHomeRetnSet
      AND     B0E21  ; Manual  ModeLampNotching
      LD      M1336  ; NotchingPressAllDown At
      ANI     D19.5
      AND     B0E23  ; Auto    ModeLampNotching
      ORB
      AND     T296  ; NotchingPress DnEnable
      ANI     M1261  ; NotchingPress #6Dn Ok
      ANI     Y2A2  ; NotchingPress #6Up Sv
      OUT     Y2A3  ; NotchingPress #6Dn Sv
981   LDI     B2A4  ; NotchingPress #7Up Sw
      ANI     B240  ; NotchingPressAllUp Sw
      ANI     M1252  ; NotchingPressAllUp Hm
      INV
      AND     B0E21  ; Manual  ModeLampNotching
      LD      M1344  ; NotchingPress   Up At
      AND     B0E23  ; Auto    ModeLampNotching
      ORB
      LDI     T308  ; NotchingPress #7Up Tm
      ORI     SM401  ; Normal  Off
      ANB
      ANI     Y2A5  ; NotchingPress #7Dn Sv
      OUT     Y2A4  ; NotchingPress #7Up Sv
994   LDI     B2A5  ; NotchingPress #7Dn Sw
      ANI     B241  ; NotchingPressAllDn Sw
      INV
      ANI     M1250  ; NotchingHomeRetnSet
      AND     B0E21  ; Manual  ModeLampNotching
      LD      M1336  ; NotchingPressAllDown At
      ANI     D19.6
      AND     B0E23  ; Auto    ModeLampNotching
      ORB
      AND     T296  ; NotchingPress DnEnable
      ANI     M1262  ; NotchingPress #7Dn Ok
      ANI     Y2A4  ; NotchingPress #7Up Sv
      OUT     Y2A5  ; NotchingPress #7Dn Sv
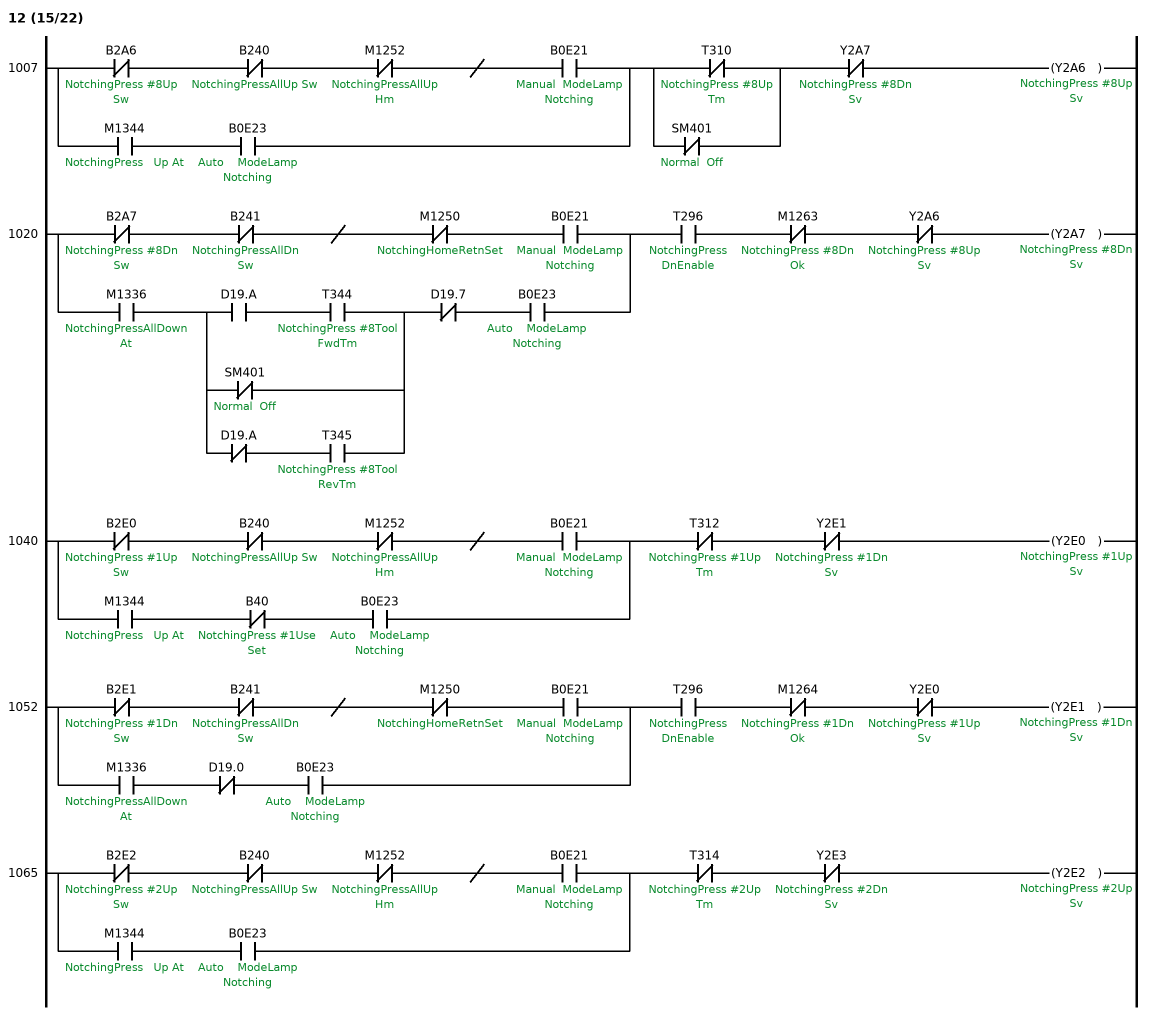
1007  LDI     B2A6  ; NotchingPress #8Up Sw
      ANI     B240  ; NotchingPressAllUp Sw
      ANI     M1252  ; NotchingPressAllUp Hm
      INV
      AND     B0E21  ; Manual  ModeLampNotching
      LD      M1344  ; NotchingPress   Up At
      AND     B0E23  ; Auto    ModeLampNotching
      ORB
      LDI     T310  ; NotchingPress #8Up Tm
      ORI     SM401  ; Normal  Off
      ANB
      ANI     Y2A7  ; NotchingPress #8Dn Sv
      OUT     Y2A6  ; NotchingPress #8Up Sv
1020  LDI     B2A7  ; NotchingPress #8Dn Sw
      ANI     B241  ; NotchingPressAllDn Sw
      INV
      ANI     M1250  ; NotchingHomeRetnSet
      AND     B0E21  ; Manual  ModeLampNotching
      LD      M1336  ; NotchingPressAllDown At
      LD      D19.A
      AND     T344  ; NotchingPress #8Tool FwdTm
      ORI     SM401  ; Normal  Off
      LDI     D19.A
      AND     T345  ; NotchingPress #8Tool RevTm
      ORB
      ANB
      ANI     D19.7
      AND     B0E23  ; Auto    ModeLampNotching
      ORB
      AND     T296  ; NotchingPress DnEnable
      ANI     M1263  ; NotchingPress #8Dn Ok
      ANI     Y2A6  ; NotchingPress #8Up Sv
      OUT     Y2A7  ; NotchingPress #8Dn Sv
1040  LDI     B2E0  ; NotchingPress #1Up Sw
      ANI     B240  ; NotchingPressAllUp Sw
      ANI     M1252  ; NotchingPressAllUp Hm
      INV
      AND     B0E21  ; Manual  ModeLampNotching
      LD      M1344  ; NotchingPress   Up At
      ANI     B40  ; NotchingPress #1Use Set
      AND     B0E23  ; Auto    ModeLampNotching
      ORB
      ANI     T312  ; NotchingPress #1Up Tm
      ANI     Y2E1  ; NotchingPress #1Dn Sv
      OUT     Y2E0  ; NotchingPress #1Up Sv
1052  LDI     B2E1  ; NotchingPress #1Dn Sw
      ANI     B241  ; NotchingPressAllDn Sw
      INV
      ANI     M1250  ; NotchingHomeRetnSet
      AND     B0E21  ; Manual  ModeLampNotching
      LD      M1336  ; NotchingPressAllDown At
      ANI     D19.0
      AND     B0E23  ; Auto    ModeLampNotching
      ORB
      AND     T296  ; NotchingPress DnEnable
      ANI     M1264  ; NotchingPress #1Dn Ok
      ANI     Y2E0  ; NotchingPress #1Up Sv
      OUT     Y2E1  ; NotchingPress #1Dn Sv
1065  LDI     B2E2  ; NotchingPress #2Up Sw
      ANI     B240  ; NotchingPressAllUp Sw
      ANI     M1252  ; NotchingPressAllUp Hm
      INV
      AND     B0E21  ; Manual  ModeLampNotching
      LD      M1344  ; NotchingPress   Up At
      AND     B0E23  ; Auto    ModeLampNotching
      ORB
      ANI     T314  ; NotchingPress #2Up Tm
      ANI     Y2E3  ; NotchingPress #2Dn Sv
      OUT     Y2E2  ; NotchingPress #2Up Sv
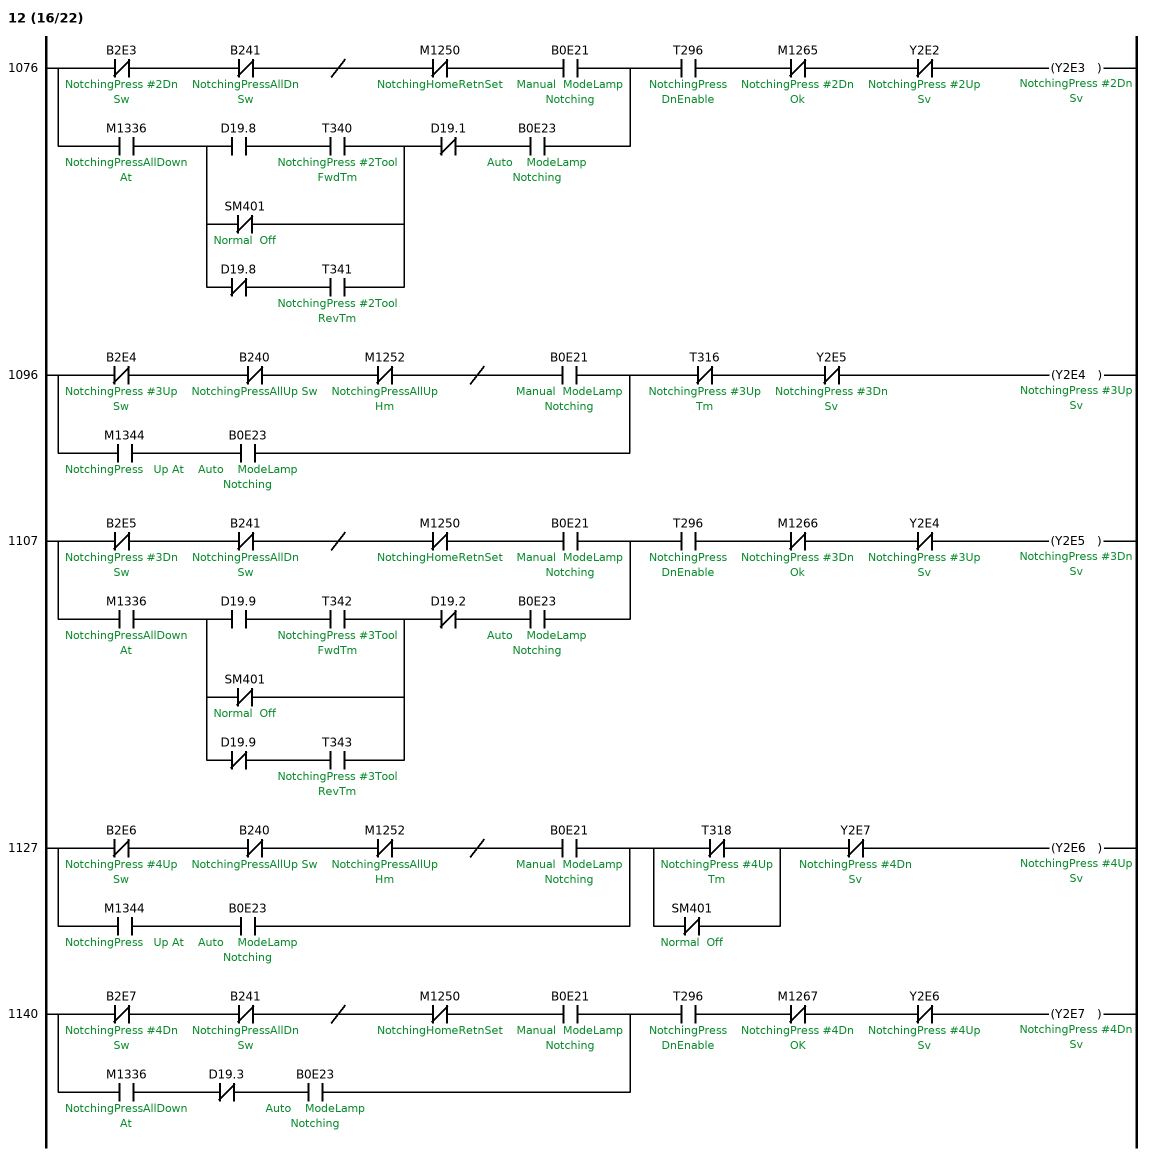
1076  LDI     B2E3  ; NotchingPress #2Dn Sw
      ANI     B241  ; NotchingPressAllDn Sw
      INV
      ANI     M1250  ; NotchingHomeRetnSet
      AND     B0E21  ; Manual  ModeLampNotching
      LD      M1336  ; NotchingPressAllDown At
      LD      D19.8
      AND     T340  ; NotchingPress #2Tool FwdTm
      ORI     SM401  ; Normal  Off
      LDI     D19.8
      AND     T341  ; NotchingPress #2Tool RevTm
      ORB
      ANB
      ANI     D19.1
      AND     B0E23  ; Auto    ModeLampNotching
      ORB
      AND     T296  ; NotchingPress DnEnable
      ANI     M1265  ; NotchingPress #2Dn Ok
      ANI     Y2E2  ; NotchingPress #2Up Sv
      OUT     Y2E3  ; NotchingPress #2Dn Sv
1096  LDI     B2E4  ; NotchingPress #3Up Sw
      ANI     B240  ; NotchingPressAllUp Sw
      ANI     M1252  ; NotchingPressAllUp Hm
      INV
      AND     B0E21  ; Manual  ModeLampNotching
      LD      M1344  ; NotchingPress   Up At
      AND     B0E23  ; Auto    ModeLampNotching
      ORB
      ANI     T316  ; NotchingPress #3Up Tm
      ANI     Y2E5  ; NotchingPress #3Dn Sv
      OUT     Y2E4  ; NotchingPress #3Up Sv
1107  LDI     B2E5  ; NotchingPress #3Dn Sw
      ANI     B241  ; NotchingPressAllDn Sw
      INV
      ANI     M1250  ; NotchingHomeRetnSet
      AND     B0E21  ; Manual  ModeLampNotching
      LD      M1336  ; NotchingPressAllDown At
      LD      D19.9
      AND     T342  ; NotchingPress #3Tool FwdTm
      ORI     SM401  ; Normal  Off
      LDI     D19.9
      AND     T343  ; NotchingPress #3Tool RevTm
      ORB
      ANB
      ANI     D19.2
      AND     B0E23  ; Auto    ModeLampNotching
      ORB
      AND     T296  ; NotchingPress DnEnable
      ANI     M1266  ; NotchingPress #3Dn Ok
      ANI     Y2E4  ; NotchingPress #3Up Sv
      OUT     Y2E5  ; NotchingPress #3Dn Sv
1127  LDI     B2E6  ; NotchingPress #4Up Sw
      ANI     B240  ; NotchingPressAllUp Sw
      ANI     M1252  ; NotchingPressAllUp Hm
      INV
      AND     B0E21  ; Manual  ModeLampNotching
      LD      M1344  ; NotchingPress   Up At
      AND     B0E23  ; Auto    ModeLampNotching
      ORB
      LDI     T318  ; NotchingPress #4Up Tm
      ORI     SM401  ; Normal  Off
      ANB
      ANI     Y2E7  ; NotchingPress #4Dn Sv
      OUT     Y2E6  ; NotchingPress #4Up Sv
1140  LDI     B2E7  ; NotchingPress #4Dn Sw
      ANI     B241  ; NotchingPressAllDn Sw
      INV
      ANI     M1250  ; NotchingHomeRetnSet
      AND     B0E21  ; Manual  ModeLampNotching
      LD      M1336  ; NotchingPressAllDown At
      ANI     D19.3
      AND     B0E23  ; Auto    ModeLampNotching
      ORB
      AND     T296  ; NotchingPress DnEnable
      ANI     M1267  ; NotchingPress #4Dn OK
      ANI     Y2E6  ; NotchingPress #4Up Sv
      OUT     Y2E7  ; NotchingPress #4Dn Sv
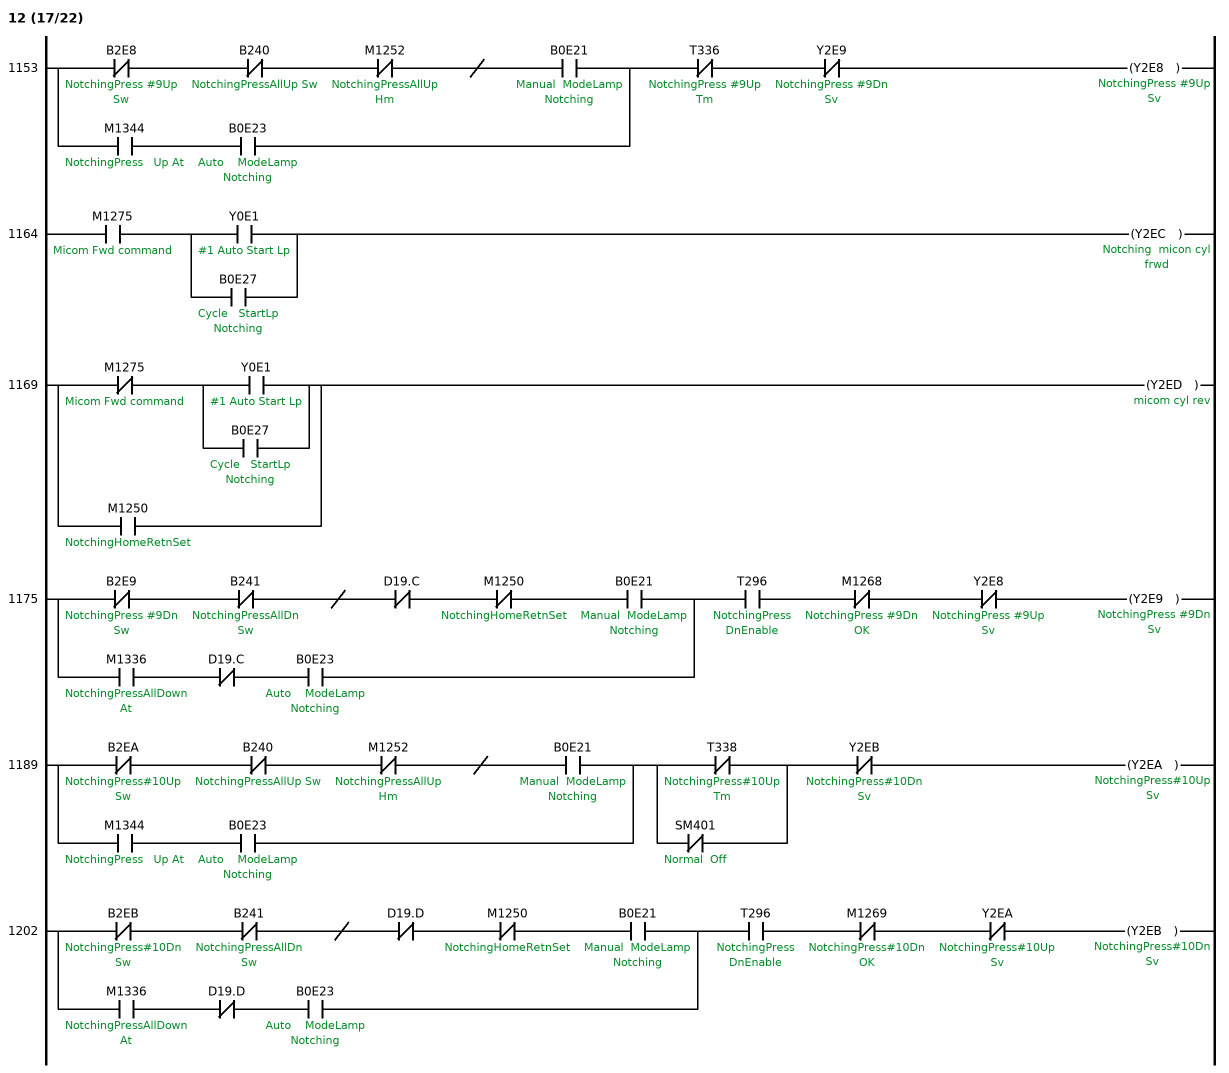
1153  LDI     B2E8  ; NotchingPress #9Up Sw
      ANI     B240  ; NotchingPressAllUp Sw
      ANI     M1252  ; NotchingPressAllUp Hm
      INV
      AND     B0E21  ; Manual  ModeLampNotching
      LD      M1344  ; NotchingPress   Up At
      AND     B0E23  ; Auto    ModeLampNotching
      ORB
      ANI     T336  ; NotchingPress #9Up Tm
      ANI     Y2E9  ; NotchingPress #9Dn Sv
      OUT     Y2E8  ; NotchingPress #9Up Sv
1164  LD      M1275  ; Micom Fwd command
      LD      Y0E1  ; #1 Auto Start Lp
      OR      B0E27  ; Cycle   StartLp Notching
      ANB
      OUT     Y2EC  ; Notching  micon cyl frwd
1169  LDI     M1275  ; Micom Fwd command
      LD      Y0E1  ; #1 Auto Start Lp
      OR      B0E27  ; Cycle   StartLp Notching
      ANB
      OR      M1250  ; NotchingHomeRetnSet
      OUT     Y2ED  ; micom cyl rev
1175  LDI     B2E9  ; NotchingPress #9Dn Sw
      ANI     B241  ; NotchingPressAllDn Sw
      INV
      ANI     D19.C
      ANI     M1250  ; NotchingHomeRetnSet
      AND     B0E21  ; Manual  ModeLampNotching
      LD      M1336  ; NotchingPressAllDown At
      ANI     D19.C
      AND     B0E23  ; Auto    ModeLampNotching
      ORB
      AND     T296  ; NotchingPress DnEnable
      ANI     M1268  ; NotchingPress #9Dn OK
      ANI     Y2E8  ; NotchingPress #9Up Sv
      OUT     Y2E9  ; NotchingPress #9Dn Sv
1189  LDI     B2EA  ; NotchingPress#10Up Sw
      ANI     B240  ; NotchingPressAllUp Sw
      ANI     M1252  ; NotchingPressAllUp Hm
      INV
      AND     B0E21  ; Manual  ModeLampNotching
      LD      M1344  ; NotchingPress   Up At
      AND     B0E23  ; Auto    ModeLampNotching
      ORB
      LDI     T338  ; NotchingPress#10Up Tm
      ORI     SM401  ; Normal  Off
      ANB
      ANI     Y2EB  ; NotchingPress#10Dn Sv
      OUT     Y2EA  ; NotchingPress#10Up Sv
1202  LDI     B2EB  ; NotchingPress#10Dn Sw
      ANI     B241  ; NotchingPressAllDn Sw
      INV
      ANI     D19.D
      ANI     M1250  ; NotchingHomeRetnSet
      AND     B0E21  ; Manual  ModeLampNotching
      LD      M1336  ; NotchingPressAllDown At
      ANI     D19.D
      AND     B0E23  ; Auto    ModeLampNotching
      ORB
      AND     T296  ; NotchingPress DnEnable
      ANI     M1269  ; NotchingPress#10Dn OK
      ANI     Y2EA  ; NotchingPress#10Up Sv
      OUT     Y2EB  ; NotchingPress#10Dn Sv
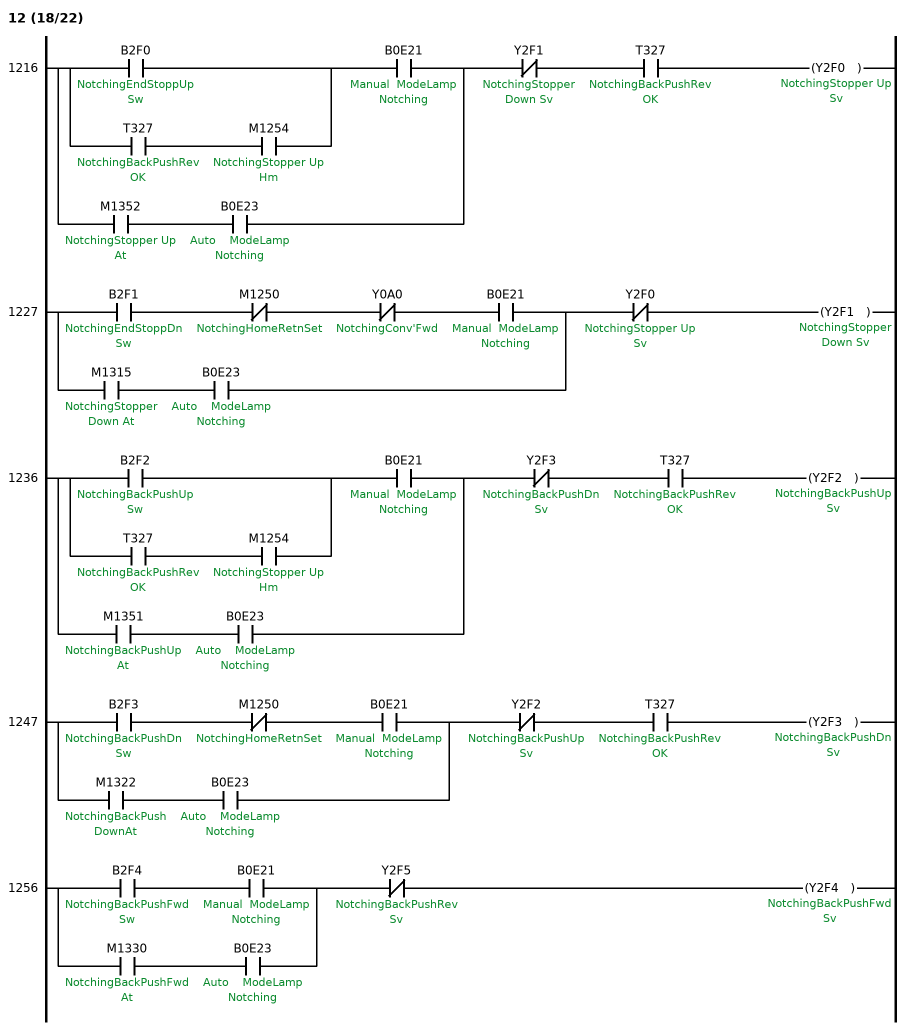
1216  LD      B2F0  ; NotchingEndStoppUpSw
      LD      T327  ; NotchingBackPushRev OK
      AND     M1254  ; NotchingStopper Up Hm
      ORB
      AND     B0E21  ; Manual  ModeLampNotching
      LD      M1352  ; NotchingStopper Up At
      AND     B0E23  ; Auto    ModeLampNotching
      ORB
      ANI     Y2F1  ; NotchingStopper Down Sv
      AND     T327  ; NotchingBackPushRev OK
      OUT     Y2F0  ; NotchingStopper Up Sv
1227  LD      B2F1  ; NotchingEndStoppDnSw
      ANI     M1250  ; NotchingHomeRetnSet
      ANI     Y0A0  ; NotchingConv'Fwd
      AND     B0E21  ; Manual  ModeLampNotching
      LD      M1315  ; NotchingStopper Down At
      AND     B0E23  ; Auto    ModeLampNotching
      ORB
      ANI     Y2F0  ; NotchingStopper Up Sv
      OUT     Y2F1  ; NotchingStopper Down Sv
1236  LD      B2F2  ; NotchingBackPushUpSw
      LD      T327  ; NotchingBackPushRev OK
      AND     M1254  ; NotchingStopper Up Hm
      ORB
      AND     B0E21  ; Manual  ModeLampNotching
      LD      M1351  ; NotchingBackPushUp At
      AND     B0E23  ; Auto    ModeLampNotching
      ORB
      ANI     Y2F3  ; NotchingBackPushDnSv
      AND     T327  ; NotchingBackPushRev OK
      OUT     Y2F2  ; NotchingBackPushUpSv
1247  LD      B2F3  ; NotchingBackPushDnSw
      ANI     M1250  ; NotchingHomeRetnSet
      AND     B0E21  ; Manual  ModeLampNotching
      LD      M1322  ; NotchingBackPushDownAt
      AND     B0E23  ; Auto    ModeLampNotching
      ORB
      ANI     Y2F2  ; NotchingBackPushUpSv
      AND     T327  ; NotchingBackPushRev OK
      OUT     Y2F3  ; NotchingBackPushDnSv
1256  LD      B2F4  ; NotchingBackPushFwdSw
      AND     B0E21  ; Manual  ModeLampNotching
      LD      M1330  ; NotchingBackPushFwdAt
      AND     B0E23  ; Auto    ModeLampNotching
      ORB
      ANI     Y2F5  ; NotchingBackPushRevSv
      OUT     Y2F4  ; NotchingBackPushFwdSv
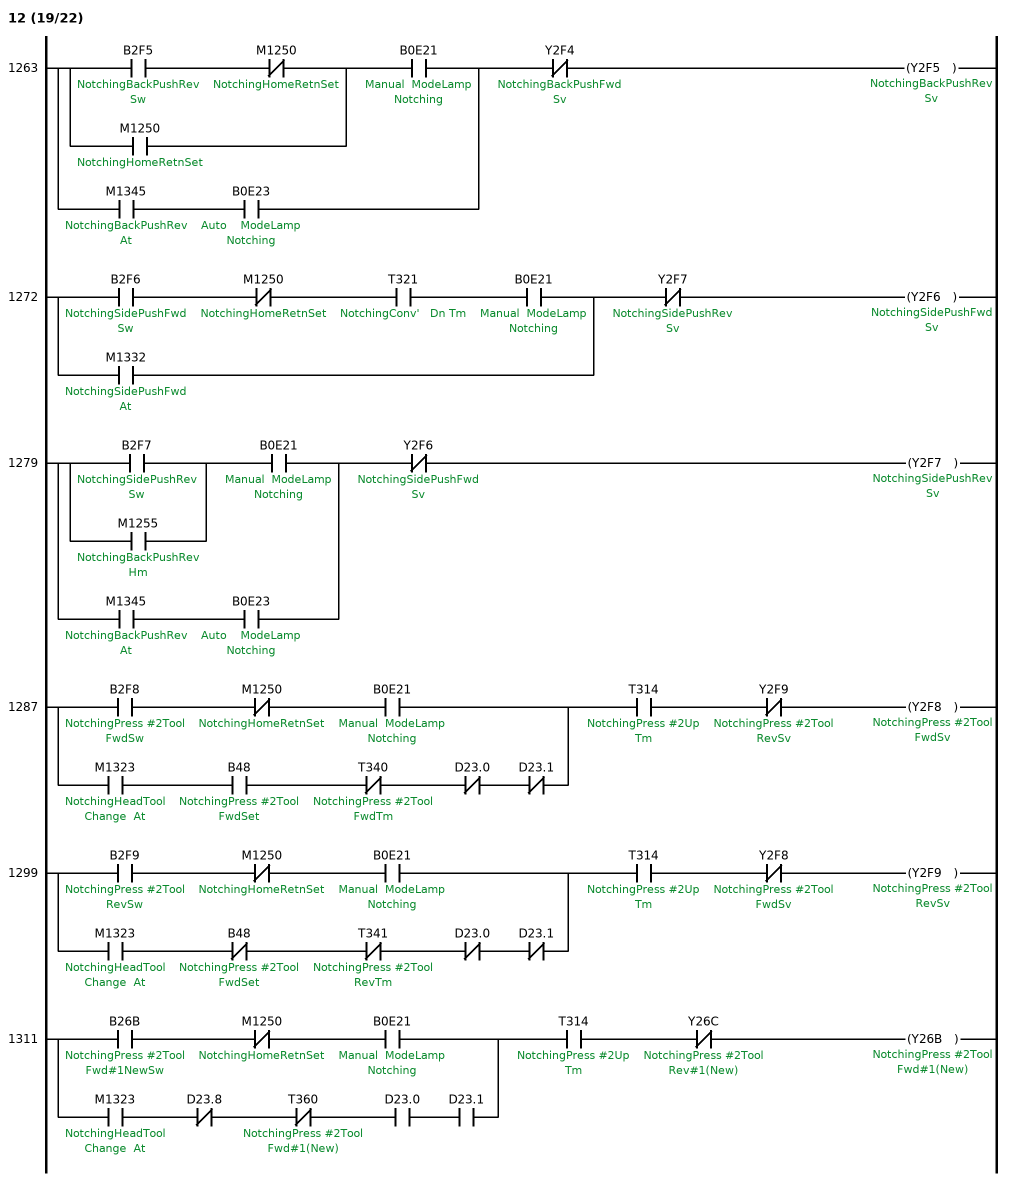
1263  LD      B2F5  ; NotchingBackPushRevSw
      ANI     M1250  ; NotchingHomeRetnSet
      OR      M1250  ; NotchingHomeRetnSet
      AND     B0E21  ; Manual  ModeLampNotching
      LD      M1345  ; NotchingBackPushRev At
      AND     B0E23  ; Auto    ModeLampNotching
      ORB
      ANI     Y2F4  ; NotchingBackPushFwdSv
      OUT     Y2F5  ; NotchingBackPushRevSv
1272  LD      B2F6  ; NotchingSidePushFwd Sw
      ANI     M1250  ; NotchingHomeRetnSet
      AND     T321  ; NotchingConv'   Dn Tm
      AND     B0E21  ; Manual  ModeLampNotching
      OR      M1332  ; NotchingSidePushFwdAt
      ANI     Y2F7  ; NotchingSidePushRev Sv
      OUT     Y2F6  ; NotchingSidePushFwd Sv
1279  LD      B2F7  ; NotchingSidePushRev Sw
      OR      M1255  ; NotchingBackPushRev Hm
      AND     B0E21  ; Manual  ModeLampNotching
      LD      M1345  ; NotchingBackPushRev At
      AND     B0E23  ; Auto    ModeLampNotching
      ORB
      ANI     Y2F6  ; NotchingSidePushFwd Sv
      OUT     Y2F7  ; NotchingSidePushRev Sv
1287  LD      B2F8  ; NotchingPress #2Tool FwdSw
      ANI     M1250  ; NotchingHomeRetnSet
      AND     B0E21  ; Manual  ModeLampNotching
      LD      M1323  ; NotchingHeadToolChange  At
      AND     B48  ; NotchingPress #2Tool FwdSet
      ANI     T340  ; NotchingPress #2Tool FwdTm
      ANI     D23.0
      ANI     D23.1
      ORB
      AND     T314  ; NotchingPress #2Up Tm
      ANI     Y2F9  ; NotchingPress #2Tool RevSv
      OUT     Y2F8  ; NotchingPress #2Tool FwdSv
1299  LD      B2F9  ; NotchingPress #2Tool RevSw
      ANI     M1250  ; NotchingHomeRetnSet
      AND     B0E21  ; Manual  ModeLampNotching
      LD      M1323  ; NotchingHeadToolChange  At
      ANI     B48  ; NotchingPress #2Tool FwdSet
      ANI     T341  ; NotchingPress #2Tool RevTm
      ANI     D23.0
      ANI     D23.1
      ORB
      AND     T314  ; NotchingPress #2Up Tm
      ANI     Y2F8  ; NotchingPress #2Tool FwdSv
      OUT     Y2F9  ; NotchingPress #2Tool RevSv
1311  LD      B26B  ; NotchingPress #2Tool Fwd#1NewSw
      ANI     M1250  ; NotchingHomeRetnSet
      AND     B0E21  ; Manual  ModeLampNotching
      LD      M1323  ; NotchingHeadToolChange  At
      ANI     D23.8
      ANI     T360  ; NotchingPress #2Tool Fwd#1(New)
      AND     D23.0
      AND     D23.1
      ORB
      AND     T314  ; NotchingPress #2Up Tm
      ANI     Y26C  ; NotchingPress #2Tool Rev#1(New)
      OUT     Y26B  ; NotchingPress #2Tool Fwd#1(New)
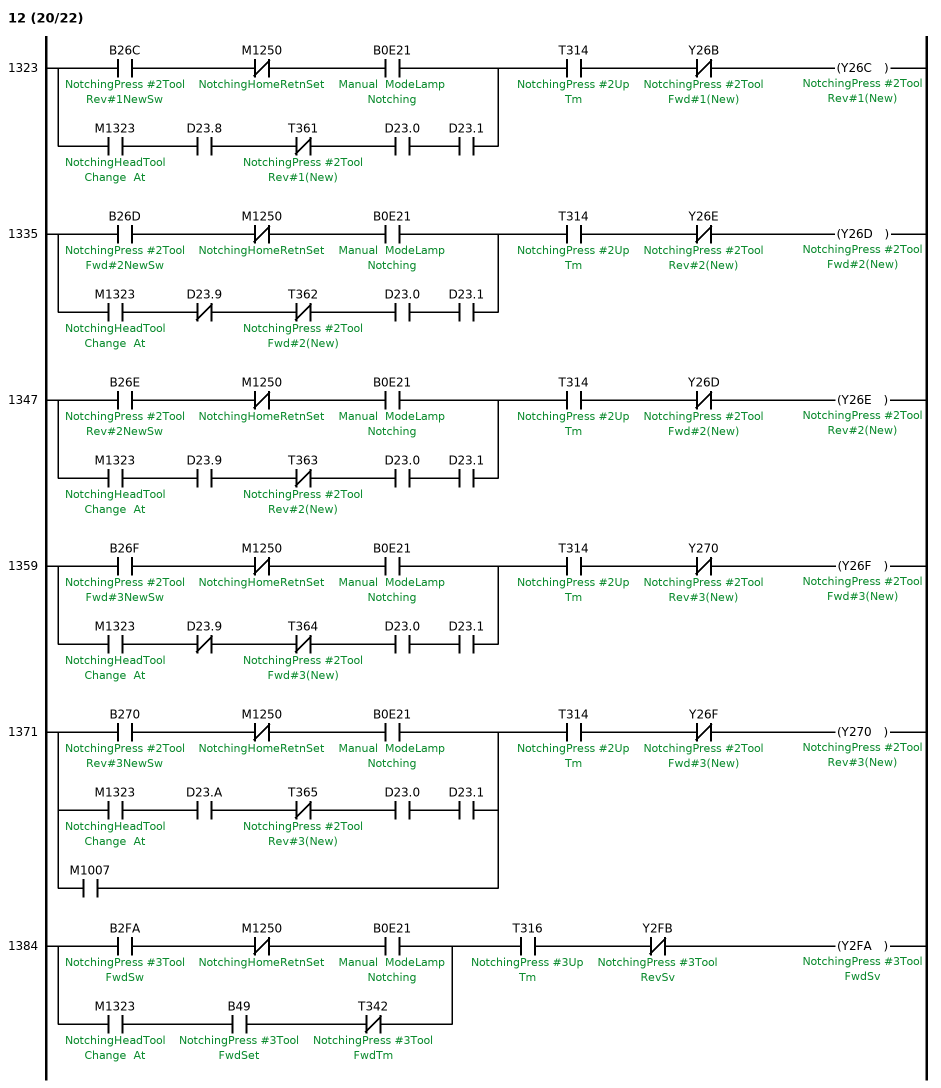
1323  LD      B26C  ; NotchingPress #2Tool Rev#1NewSw
      ANI     M1250  ; NotchingHomeRetnSet
      AND     B0E21  ; Manual  ModeLampNotching
      LD      M1323  ; NotchingHeadToolChange  At
      AND     D23.8
      ANI     T361  ; NotchingPress #2Tool Rev#1(New)
      AND     D23.0
      AND     D23.1
      ORB
      AND     T314  ; NotchingPress #2Up Tm
      ANI     Y26B  ; NotchingPress #2Tool Fwd#1(New)
      OUT     Y26C  ; NotchingPress #2Tool Rev#1(New)
1335  LD      B26D  ; NotchingPress #2Tool Fwd#2NewSw
      ANI     M1250  ; NotchingHomeRetnSet
      AND     B0E21  ; Manual  ModeLampNotching
      LD      M1323  ; NotchingHeadToolChange  At
      ANI     D23.9
      ANI     T362  ; NotchingPress #2Tool Fwd#2(New)
      AND     D23.0
      AND     D23.1
      ORB
      AND     T314  ; NotchingPress #2Up Tm
      ANI     Y26E  ; NotchingPress #2Tool Rev#2(New)
      OUT     Y26D  ; NotchingPress #2Tool Fwd#2(New)
1347  LD      B26E  ; NotchingPress #2Tool Rev#2NewSw
      ANI     M1250  ; NotchingHomeRetnSet
      AND     B0E21  ; Manual  ModeLampNotching
      LD      M1323  ; NotchingHeadToolChange  At
      AND     D23.9
      ANI     T363  ; NotchingPress #2Tool Rev#2(New)
      AND     D23.0
      AND     D23.1
      ORB
      AND     T314  ; NotchingPress #2Up Tm
      ANI     Y26D  ; NotchingPress #2Tool Fwd#2(New)
      OUT     Y26E  ; NotchingPress #2Tool Rev#2(New)
1359  LD      B26F  ; NotchingPress #2Tool Fwd#3NewSw
      ANI     M1250  ; NotchingHomeRetnSet
      AND     B0E21  ; Manual  ModeLampNotching
      LD      M1323  ; NotchingHeadToolChange  At
      ANI     D23.9
      ANI     T364  ; NotchingPress #2Tool Fwd#3(New)
      AND     D23.0
      AND     D23.1
      ORB
      AND     T314  ; NotchingPress #2Up Tm
      ANI     Y270  ; NotchingPress #2Tool Rev#3(New)
      OUT     Y26F  ; NotchingPress #2Tool Fwd#3(New)
1371  LD      B270  ; NotchingPress #2Tool Rev#3NewSw
      ANI     M1250  ; NotchingHomeRetnSet
      AND     B0E21  ; Manual  ModeLampNotching
      LD      M1323  ; NotchingHeadToolChange  At
      AND     D23.A
      ANI     T365  ; NotchingPress #2Tool Rev#3(New)
      AND     D23.0
      AND     D23.1
      ORB
      OR      M1007
      AND     T314  ; NotchingPress #2Up Tm
      ANI     Y26F  ; NotchingPress #2Tool Fwd#3(New)
      OUT     Y270  ; NotchingPress #2Tool Rev#3(New)
1384  LD      B2FA  ; NotchingPress #3Tool FwdSw
      ANI     M1250  ; NotchingHomeRetnSet
      AND     B0E21  ; Manual  ModeLampNotching
      LD      M1323  ; NotchingHeadToolChange  At
      AND     B49  ; NotchingPress #3Tool FwdSet
      ANI     T342  ; NotchingPress #3Tool FwdTm
      ORB
      AND     T316  ; NotchingPress #3Up Tm
      ANI     Y2FB  ; NotchingPress #3Tool RevSv
      OUT     Y2FA  ; NotchingPress #3Tool FwdSv
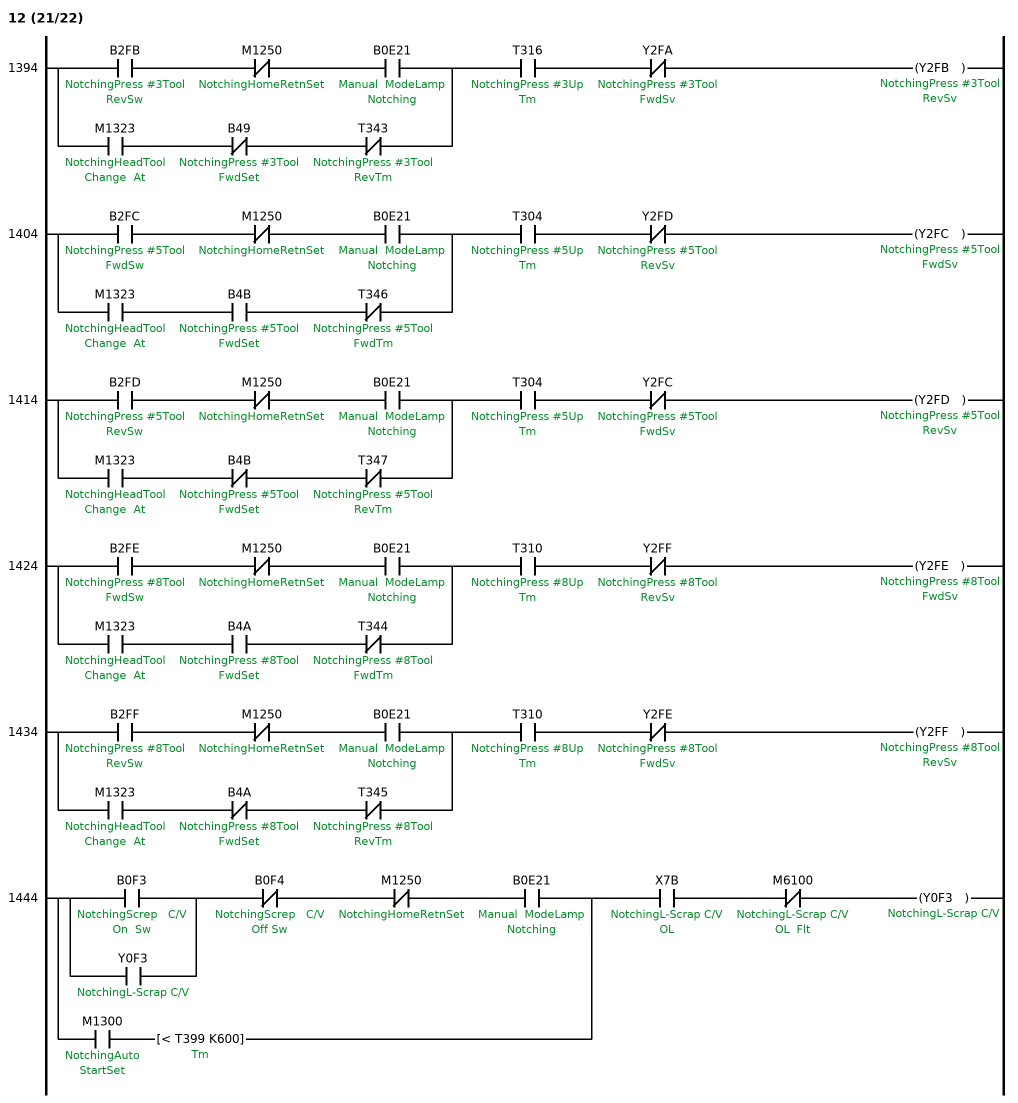
1394  LD      B2FB  ; NotchingPress #3Tool RevSw
      ANI     M1250  ; NotchingHomeRetnSet
      AND     B0E21  ; Manual  ModeLampNotching
      LD      M1323  ; NotchingHeadToolChange  At
      ANI     B49  ; NotchingPress #3Tool FwdSet
      ANI     T343  ; NotchingPress #3Tool RevTm
      ORB
      AND     T316  ; NotchingPress #3Up Tm
      ANI     Y2FA  ; NotchingPress #3Tool FwdSv
      OUT     Y2FB  ; NotchingPress #3Tool RevSv
1404  LD      B2FC  ; NotchingPress #5Tool FwdSw
      ANI     M1250  ; NotchingHomeRetnSet
      AND     B0E21  ; Manual  ModeLampNotching
      LD      M1323  ; NotchingHeadToolChange  At
      AND     B4B  ; NotchingPress #5Tool FwdSet
      ANI     T346  ; NotchingPress #5Tool FwdTm
      ORB
      AND     T304  ; NotchingPress #5Up Tm
      ANI     Y2FD  ; NotchingPress #5Tool RevSv
      OUT     Y2FC  ; NotchingPress #5Tool FwdSv
1414  LD      B2FD  ; NotchingPress #5Tool RevSw
      ANI     M1250  ; NotchingHomeRetnSet
      AND     B0E21  ; Manual  ModeLampNotching
      LD      M1323  ; NotchingHeadToolChange  At
      ANI     B4B  ; NotchingPress #5Tool FwdSet
      ANI     T347  ; NotchingPress #5Tool RevTm
      ORB
      AND     T304  ; NotchingPress #5Up Tm
      ANI     Y2FC  ; NotchingPress #5Tool FwdSv
      OUT     Y2FD  ; NotchingPress #5Tool RevSv
1424  LD      B2FE  ; NotchingPress #8Tool FwdSw
      ANI     M1250  ; NotchingHomeRetnSet
      AND     B0E21  ; Manual  ModeLampNotching
      LD      M1323  ; NotchingHeadToolChange  At
      AND     B4A  ; NotchingPress #8Tool FwdSet
      ANI     T344  ; NotchingPress #8Tool FwdTm
      ORB
      AND     T310  ; NotchingPress #8Up Tm
      ANI     Y2FF  ; NotchingPress #8Tool RevSv
      OUT     Y2FE  ; NotchingPress #8Tool FwdSv
1434  LD      B2FF  ; NotchingPress #8Tool RevSw
      ANI     M1250  ; NotchingHomeRetnSet
      AND     B0E21  ; Manual  ModeLampNotching
      LD      M1323  ; NotchingHeadToolChange  At
      ANI     B4A  ; NotchingPress #8Tool FwdSet
      ANI     T345  ; NotchingPress #8Tool RevTm
      ORB
      AND     T310  ; NotchingPress #8Up Tm
      ANI     Y2FE  ; NotchingPress #8Tool FwdSv
      OUT     Y2FF  ; NotchingPress #8Tool RevSv
1444  LD      B0F3  ; NotchingScrep   C/V On  Sw
      OR      Y0F3  ; NotchingL-Scrap C/V
      ANI     B0F4  ; NotchingScrep   C/V Off Sw
      ANI     M1250  ; NotchingHomeRetnSet
      AND     B0E21  ; Manual  ModeLampNotching
      LD      M1300  ; NotchingAuto    StartSet
      AND<    T399 K600  ; Tm
      ORB
      AND     X7B  ; NotchingL-Scrap C/V OL
      ANI     M6100  ; NotchingL-Scrap C/V OL  Flt
      OUT     Y0F3  ; NotchingL-Scrap C/V
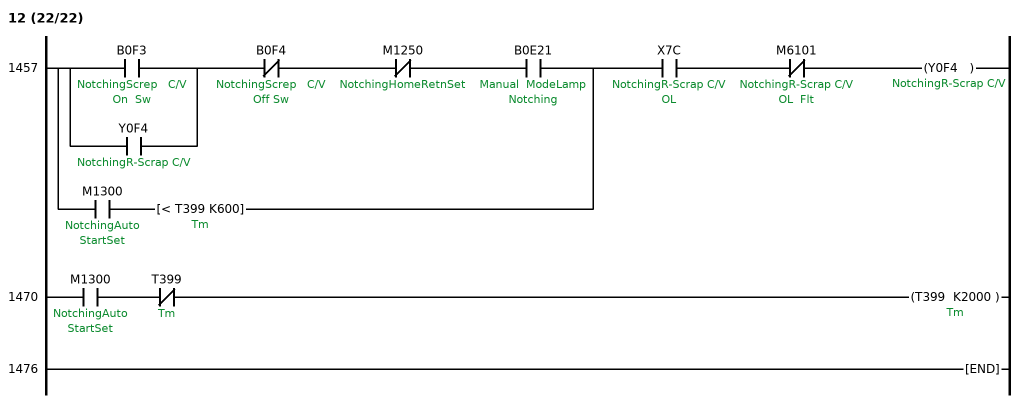
1457  LD      B0F3  ; NotchingScrep   C/V On  Sw
      OR      Y0F4  ; NotchingR-Scrap C/V
      ANI     B0F4  ; NotchingScrep   C/V Off Sw
      ANI     M1250  ; NotchingHomeRetnSet
      AND     B0E21  ; Manual  ModeLampNotching
      LD      M1300  ; NotchingAuto    StartSet
      AND<    T399 K600  ; Tm
      ORB
      AND     X7C  ; NotchingR-Scrap C/V OL
      ANI     M6101  ; NotchingR-Scrap C/V OL  Flt
      OUT     Y0F4  ; NotchingR-Scrap C/V
1470  LD      M1300  ; NotchingAuto    StartSet
      ANI     T399  ; Tm
      OUT     T399 K2000  ; Tm
1476  END
END_PROGRAM

PROGRAM 13  // Idle Conveyor
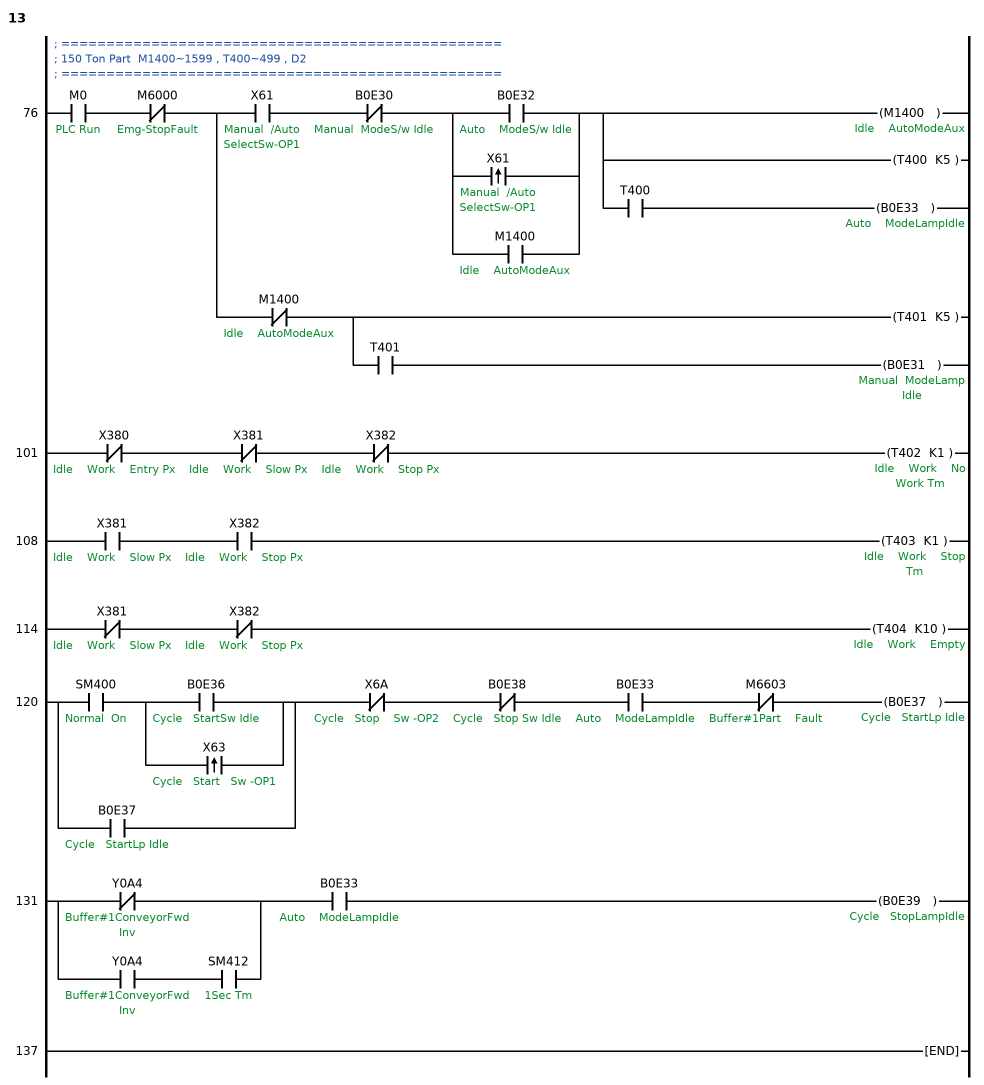
; =================================================
; 150 Ton Part  M1400~1599 , T400~499 , D2
; =================================================
76    LD      M0  ; PLC Run
      ANI     M6000  ; Emg-StopFault
      MPS
      AND     X61  ; Manual  /Auto   SelectSw-OP1
      ANI     B0E30  ; Manual  ModeS/w Idle
      LD      B0E32  ; Auto    ModeS/w Idle
      ORP     X61  ; Manual  /Auto   SelectSw-OP1
      OR      M1400  ; Idle    AutoModeAux
      ANB
      OUT     M1400  ; Idle    AutoModeAux
      OUT     T400 K5
      AND     T400
      OUT     B0E33  ; Auto    ModeLampIdle
      MPP
      ANI     M1400  ; Idle    AutoModeAux
      OUT     T401 K5
      AND     T401
      OUT     B0E31  ; Manual  ModeLampIdle
101   LDI     X380  ; Idle    Work    Entry Px
      ANI     X381  ; Idle    Work    Slow Px
      ANI     X382  ; Idle    Work    Stop Px
      OUT     T402 K1  ; Idle    Work    No Work Tm
108   LD      X381  ; Idle    Work    Slow Px
      AND     X382  ; Idle    Work    Stop Px
      OUT     T403 K1  ; Idle    Work    Stop Tm
114   LDI     X381  ; Idle    Work    Slow Px
      ANI     X382  ; Idle    Work    Stop Px
      OUT     T404 K10  ; Idle    Work    Empty
120   LD      SM400  ; Normal  On
      LD      B0E36  ; Cycle   StartSw Idle
      ORP     X63  ; Cycle   Start   Sw -OP1
      ANB
      OR      B0E37  ; Cycle   StartLp Idle
      ANI     X6A  ; Cycle   Stop    Sw -OP2
      ANI     B0E38  ; Cycle   Stop Sw Idle
      AND     B0E33  ; Auto    ModeLampIdle
      ANI     M6603  ; Buffer#1Part    Fault
      OUT     B0E37  ; Cycle   StartLp Idle
131   LDI     Y0A4  ; Buffer#1ConveyorFwd Inv
      LD      Y0A4  ; Buffer#1ConveyorFwd Inv
      AND     SM412  ; 1Sec Tm
      ORB
      AND     B0E33  ; Auto    ModeLampIdle
      OUT     B0E39  ; Cycle   StopLampIdle
137   END
END_PROGRAM

PROGRAM 14  // Turn Over
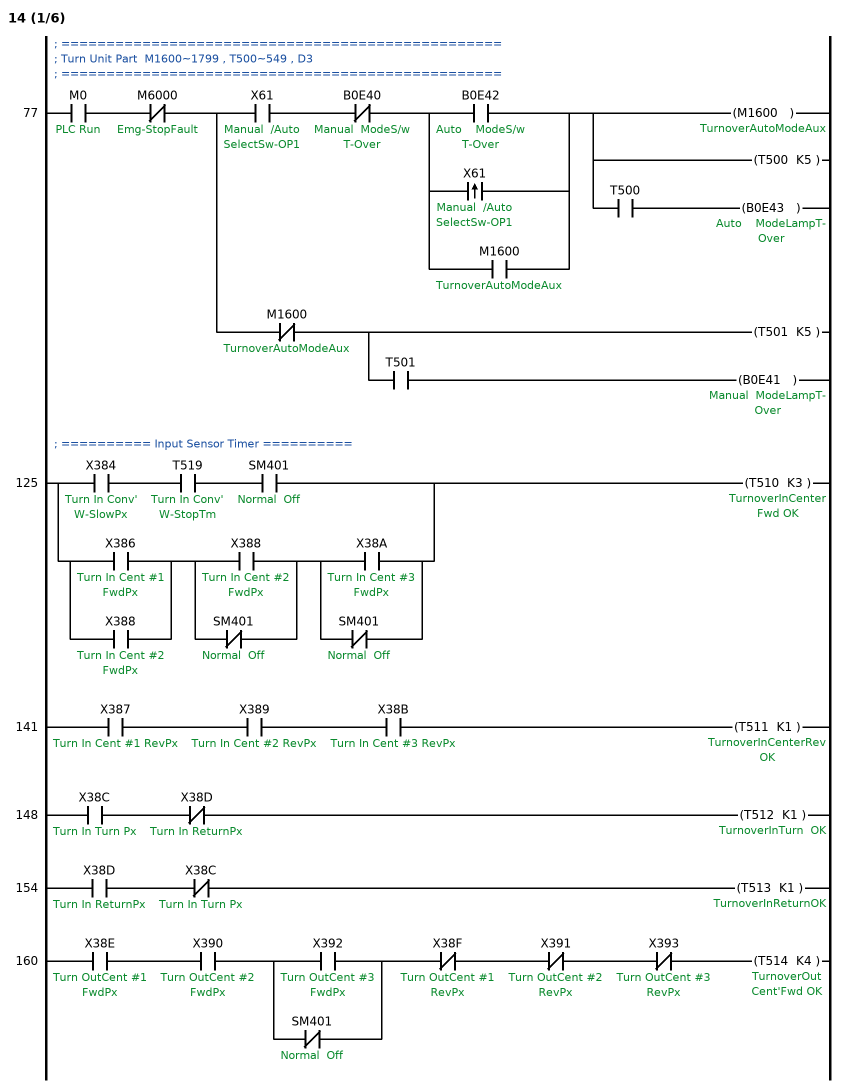
; =================================================
; Turn Unit Part  M1600~1799 , T500~549 , D3
; =================================================
77    LD      M0  ; PLC Run
      ANI     M6000  ; Emg-StopFault
      MPS
      AND     X61  ; Manual  /Auto   SelectSw-OP1
      ANI     B0E40  ; Manual  ModeS/w T-Over
      LD      B0E42  ; Auto    ModeS/w T-Over
      ORP     X61  ; Manual  /Auto   SelectSw-OP1
      OR      M1600  ; TurnoverAutoModeAux
      ANB
      OUT     M1600  ; TurnoverAutoModeAux
      OUT     T500 K5
      AND     T500
      OUT     B0E43  ; Auto    ModeLampT-Over
      MPP
      ANI     M1600  ; TurnoverAutoModeAux
      OUT     T501 K5
      AND     T501
      OUT     B0E41  ; Manual  ModeLampT-Over
; ========== Input Sensor Timer ==========
125   LD      X384  ; Turn In Conv'   W-SlowPx
      AND     T519  ; Turn In Conv'   W-StopTm
      AND     SM401  ; Normal  Off
      LD      X386  ; Turn In Cent #1 FwdPx
      OR      X388  ; Turn In Cent #2 FwdPx
      LD      X388  ; Turn In Cent #2 FwdPx
      ORI     SM401  ; Normal  Off
      ANB
      LD      X38A  ; Turn In Cent #3 FwdPx
      ORI     SM401  ; Normal  Off
      ANB
      ORB
      OUT     T510 K3  ; TurnoverInCenterFwd OK
141   LD      X387  ; Turn In Cent #1 RevPx
      AND     X389  ; Turn In Cent #2 RevPx
      AND     X38B  ; Turn In Cent #3 RevPx
      OUT     T511 K1  ; TurnoverInCenterRev OK
148   LD      X38C  ; Turn In Turn Px
      ANI     X38D  ; Turn In ReturnPx
      OUT     T512 K1  ; TurnoverInTurn  OK
154   LD      X38D  ; Turn In ReturnPx
      ANI     X38C  ; Turn In Turn Px
      OUT     T513 K1  ; TurnoverInReturnOK
160   LD      X38E  ; Turn OutCent #1 FwdPx
      AND     X390  ; Turn OutCent #2 FwdPx
      LD      X392  ; Turn OutCent #3 FwdPx
      ORI     SM401  ; Normal  Off
      ANB
      ANI     X38F  ; Turn OutCent #1 RevPx
      ANI     X391  ; Turn OutCent #2 RevPx
      ANI     X393  ; Turn OutCent #3 RevPx
      OUT     T514 K4  ; TurnoverOutCent'Fwd OK
